// TwinCAT 3 PLC project IDPLC
// ProgramVersion: 3.1.4024.12
// libraries:
//   Recipe Management, * (System)
//   Tc2_Drive, * (Beckhoff Automation GmbH)
//   Tc2_EtherCAT, * (Beckhoff Automation GmbH)
//   Tc2_Math, * (Beckhoff Automation GmbH)
//   Tc2_MC2, * (Beckhoff Automation GmbH)
//   Tc2_ModbusSrv, * (Beckhoff Automation GmbH)
//   Tc2_NC, * (Beckhoff Automation GmbH)
//   Tc2_NcDrive, * (Beckhoff Automation GmbH)
//   Tc2_Standard, * (Beckhoff Automation GmbH)
//   Tc2_System, * (Beckhoff Automation GmbH)
//   Tc2_Utilities, * (Beckhoff Automation GmbH)
//   Tc3_Module, * (Beckhoff Automation GmbH)
//   VisuDialogs, * (System)
// project tree:
//   DUTs/ DUT.TcDUT (not stored), DUT_SENSOR_DATAS_1.TcDUT (not stored), DUT_SENSOR_DATAS_h1.TcDUT, DUT_SENSOR_DATAS_h2.TcDUT, DUT_SENSOR_DATAS_h3.TcDUT, DUT_SENSOR_DATAS_h4.TcDUT, DUT_SENSOR_DATAS_h5.TcDUT, DUT_SENSOR_DATAS_h6.TcDUT, DUT_SENSOR_DATAS_h7.TcDUT, DUT_SENSOR_DATAS_h8.TcDUT, DUT_SENSOR_DATAS_8.TcDUT (not stored), DUT_SENSOR_DATAS_2.TcDUT (not stored), DUT_SENSOR_DATAS_3.TcDUT (not stored), DUT_SENSOR_DATAS_4.TcDUT (not stored), DUT_SENSOR_DATAS_5.TcDUT (not stored), DUT_SENSOR_DATAS_6.TcDUT (not stored), DUT_SENSOR_DATAS_7.TcDUT (not stored), IEEE754_Convert.TcDUT, Struct_M_Compensation.TcDUT (not stored), Struct_M_Gap2Coil.TcDUT, Struct_M_lakeshore.TcDUT (not stored), ST_P180.TcDUT (not stored), ST_P183.TcDUT (not stored), ST_P182.TcDUT (not stored)
//   / GlobalTextList.TcGTLO, PlcTask.TcTTO (not stored), RecipeManager.TcRMO (not stored), Task_Safe.TcTTO, 视图管理器.TcVMO (not stored)
//   GVLs/ Global_Variables.TcGVL, Variable_Configuration.TcGVL (not stored)
//   POUs/0.UserMode/ F_GetSysTime.TcPOU (not stored), UserMode.TcPOU
//   POUs/1.CarrierMode/GapMode/ BCGapMode.TcPOU, GapMode.TcPOU
//   POUs/1.CarrierMode/SingleCarrierMode/ SingleCarrierMode.TcPOU
//   POUs/2.SingleMotorMode/DebugMode/ DebugMode.TcPOU
//   POUs/2.SingleMotorMode/TaperMode/ TaperMode.TcPOU
//   POUs/CoilControl/ PS1.TcPOU, PS3.TcPOU, PS2.TcPOU
//   POUs/CommonFB/ExternFB/ FB_LedShow.TcPOU (not stored), FB_PlcEmergencyStop.TcPOU (not stored)
//   POUs/CommonFB/MainFB/ FB_CoupleAxis.TcPOU, FB_DecoupleAxis.TcPOU, FB_Move.TcPOU, FB_Power.TcPOU, FB_SetAxisPosition.TcPOU, FB_SetMotorAxisPosition.TcPOU, FB_Stop.TcPOU
//   POUs/ MAIN.TcPOU
//   POUs/MainPRG/ FB_CheckCoupleStatus.TcPOU (not stored)
//   POUs/TiltSensor/ FB_Simple_MovingAvg.TcPOU, SAFE.TcPOU
//   VISUs/ Visualization.TcVIS

CONFIGURATION IDPLC
    RESOURCE PLC ON TwinCAT3
        TASK Task_Safe(INTERVAL := T#1ms, PRIORITY := 1);
        PROGRAM SAFE WITH Task_Safe : SAFE;
    END_RESOURCE
END_CONFIGURATION

// ---- DUTs/DUT_SENSOR_DATAS_h1.TcDUT
TYPE DUT_SENSOR_DATAS_h1 :
UNION
	data_lreal:REAL;
	data_byte:ARRAY[0..3] OF BYTE;
END_UNION
END_TYPE

// ---- DUTs/DUT_SENSOR_DATAS_h2.TcDUT
TYPE DUT_SENSOR_DATAS_h2 :
UNION
	data_lreal:REAL;
	data_byte:ARRAY[0..3] OF BYTE;
END_UNION
END_TYPE

// ---- DUTs/DUT_SENSOR_DATAS_h3.TcDUT
TYPE DUT_SENSOR_DATAS_h3 :
UNION
	data_lreal:REAL;
	data_byte:ARRAY[0..3] OF BYTE;
END_UNION
END_TYPE

// ---- DUTs/DUT_SENSOR_DATAS_h4.TcDUT
TYPE DUT_SENSOR_DATAS_h4 :
UNION
	data_lreal:REAL;
	data_byte:ARRAY[0..3] OF BYTE;
END_UNION
END_TYPE

// ---- DUTs/DUT_SENSOR_DATAS_h5.TcDUT
TYPE DUT_SENSOR_DATAS_h5 :
UNION
	data_lreal:REAL;
	data_byte:ARRAY[0..3] OF BYTE;
END_UNION
END_TYPE

// ---- DUTs/DUT_SENSOR_DATAS_h6.TcDUT
TYPE DUT_SENSOR_DATAS_h6 :
UNION
	data_lreal:REAL;
	data_byte:ARRAY[0..3] OF BYTE;
END_UNION
END_TYPE

// ---- DUTs/DUT_SENSOR_DATAS_h7.TcDUT
TYPE DUT_SENSOR_DATAS_h7 :
UNION
	data_lreal:REAL;
	data_byte:ARRAY[0..3] OF BYTE;
END_UNION
END_TYPE

// ---- DUTs/DUT_SENSOR_DATAS_h8.TcDUT
TYPE DUT_SENSOR_DATAS_h8 :
UNION
	data_lreal:REAL;
	data_byte:ARRAY[0..3] OF BYTE;
END_UNION
END_TYPE

// ---- DUTs/IEEE754_Convert.TcDUT
TYPE IEEE754_Convert :
UNION
	data_float:REAL;
	data_word:ARRAY[0..1] OF WORD;
END_UNION
END_TYPE

// ---- DUTs/Struct_M_Gap2Coil.TcDUT
TYPE Struct_M_Gap2Coil :
STRUCT
	Gap:LREAL;
	CoilCurrent:LREAL;
END_STRUCT
END_TYPE

// ---- GVLs/Global_Variables.TcGVL
//{attribute 'Tc2GvlVarNames'}
VAR_GLOBAL
(*IDControl Ready*)
	IDControlReady:BOOL;
(*Maintenance Mode*)
	MaintenanceMode:BOOL;
	MaintenanceModeLed:BOOL;
(*RecipeDescription*)
	RecipeSavedDate:STRING;
	RecipeDescription:STRING;
(*key Command*)
	btn_Power:BOOL;
	btn_PowerOn: BOOL;
	btn_PowerOff: BOOL;
(*Reset*)
	btn_Reset:BOOL;
(*ModeStatus*)
	ModeStatus:INT;
(*Error Massage*)
	Error:BOOL;
	ErrorID:DINT;
	ErrorDescription:STRING;
(*加载配方参数*)
	LoadRecipeParameters:BOOL;
	loadParametersDone:BOOL;
(*Max Velocity Global*)
	MaxVelocityGlobalVelocity : LREAL;
(*设置光栅bias done *)	
	PositionBiasDone:BOOL;
(*回程差*)
	HysteresisError:LREAL;
(*Drive Status*)
	DriveStatus:DINT;//1:Drive Ready;2:Axis is in operation;0:Others
(*光栅漂移误差阈值*)
	LEDriftErrorThreshold:LREAL:=0.001;
(*Lag Distance threshold*)
	PosDiff_LeftTopLin: LREAL:=0.5;
	PosDiff_RightTopLin:LREAL:=0.5;
	PosDiff_LeftBottomLin:LREAL:=0.5;
	PosDiff_RightBottomLin:LREAL:=0.5;
(*UserMode Threshold*)
	Threshold_UserTopPos: LREAL:=0.5;
	Threshold_UserBottomPos: LREAL:=0.5;
	Threshold_UserLeftPos: LREAL:=0.5;
	Threshold_UserRightPos: LREAL:=0.5;
	Threshold_UserTopVelo: LREAL:=0.5;
	Threshold_UserBottomVelo: LREAL:=0.5;
	Threshold_UserLeftVelo: LREAL:=0.5;
	Threshold_UserRightVelo: LREAL:=0.5;
	//
	Range_UserTaperPos:LREAL:=4.01;
	Range_UserTaperVelo:LREAL:=1.01;
	//Diff_TaperLeftPos:LREAL:=0.01;
	//Diff_TaperLeftVelo:LREAL:=0.2;
	//Diff_TaperRightPos:LREAL:=0.05;
	//Diff_TaperRightVelo:LREAL:=0.5;
	//Taper_BeyondRangePositive:BOOL;
	//Diff_TaperTopPos:LREAL:=0.05;
	//Diff_TaperBottomPos:LREAL:=0.05;
	//Taper_BeyondRangeNegtive:BOOL;
(*BCGap Threshold*)
	Threshold_BCTopPos: LREAL:=0.5;
	Threshold_BCBottomPos: LREAL:=0.5;
	Threshold_BCLeftPos: LREAL:=0.5;
	Threshold_BCRightPos: LREAL:=0.5;
	Threshold_BCTopVelo: LREAL:=0.5;
	Threshold_BCBottomVelo: LREAL:=0.5;
	Threshold_BCLeftVelo: LREAL:=0.5;
	Threshold_BCRightVelo: LREAL:=0.5;
(*DebugMode Threshold*)
	Threshold_TopPos_Debug: LREAL:=4;
	Threshold_BottomPos_Debug: LREAL:=4;
	Threshold_LeftPos_Debug: LREAL:=4;
	Threshold_RightPos_Debug: LREAL:=4;
	//单轴目标位置和当前位置之差，阈值
	Threshold_LeftTopPos_Debug: LREAL:=0.4;	
	Threshold_RightTopPos_Debug: LREAL:=0.4;
	Threshold_LeftBottomPos_Debug: LREAL:=0.4;
	Threshold_RightBottomPos_Debug: LREAL:=0.4;
(*Taper Mode Threshold*)
	Range_TaperPos:LREAL:=5.01;
	Range_TaperVelo:LREAL:=1.01;
	Threshold_TaperLeftPos:LREAL:=0.01;
	Threshold_TaperLeftVelo:LREAL:=0.2;
	Threshold_TaperRightPos:LREAL:=0.05;
	Threshold_TaperRightVelo:LREAL:=0.5;
	Taper_BeyondRangePositive:BOOL;
	Threshold_TaperTopPos:LREAL:=0.05;
	Threshold_TaperBottomPos:LREAL:=0.05;
	Taper_BeyondRangeNegtive:BOOL;
(*SingleCarrierMode threshold*)
	Threshold_TopPos_SingleCarrier: LREAL:=2;
	Threshold_BottomPos_SingleCarrier: LREAL:=2;
	Threshold_LeftPos_SingleCarrier: LREAL:=2;
	Threshold_RightPos_SingleCarrier: LREAL:=2;
	Threshold_TopVelo_SingleCarrier: LREAL:=2;
	Threshold_BottomVelo_SingleCarrier: LREAL:=2;
	Threshold_LeftVelo_SingleCarrier: LREAL:=2;
	Threshold_RightVelo_SingleCarrier: LREAL:=2;
(*Compensation Value*)
	(*Moving or notmoving*)
	moveStatusLeftTop: BOOL;
	moveStatusRightTop: BOOL;
	moveStatusLeftBottom: BOOL;
	moveStatusRightBottom: BOOL;
	moveStatusAllAxis: BOOL;
	moveStatusAnyAxis: BOOL;
	moveStatusGap:BOOL;
	moveStatusTaper:BOOL;
(*Moving or notmoving-Motor*)
	moveStatusLeftTopMotor: BOOL;
	moveStatusRightTopMotor: BOOL;
	moveStatusLeftBottomMotor: BOOL;
	moveStatusRightBottomMotor: BOOL;
	moveStatusAllAxisMotor: BOOL;
	moveStatusAnyAxisMotor: BOOL;
	(*input protection*)
	//
	min_UserGapPositionNew:LREAL:=10;
	max_UserGapPositionNew:LREAL:=200;
	inRange_UserGapPositionNew:BOOL;
	//LE protection position
	min_UserLEProtectionGapPosition:LREAL;
	min_ThresholdGapSoft2LEProtection:LREAL;
	max_UserLEProtectionGapPosition:LREAL;
	max_ThresholdGapSoft2LEProtection:LREAL;
	//
	min_UserGapVelocityNew:LREAL:=0;
	max_UserGapVelocityNew:LREAL:=2;
	inRange_UserGapVelocityNew:BOOL;
	//
	min_UserTaperPositionNew: LREAL:=0;;
	max_UserTaperPositionNew: LREAL:=1;
	inRange_UserTaperPositionNew: BOOL;
	//
	min_UserTaperVelocityNew: LREAL:=0;
	max_UserTaperVelocityNew: LREAL:=1;
	inRange_UserTaperVelocityNew: BOOL;

	M_Compensation:ARRAY[1..18] OF Struct_M_Compensation
:=[
(Encoder:=0,	LeftTop:=0,	RightTop:=0,		LeftBottom:=0,	RightBottom:=0,	InRange:=FALSE),
(Encoder:=5.5,	LeftTop:=5.5,	RightTop:=5.5,	LeftBottom:=5.5,	RightBottom:=5.5,	InRange:=FALSE),
(Encoder:=6.0,	LeftTop:=6.0,	RightTop:=6.0,	LeftBottom:=6.0,	RightBottom:=6.0,	InRange:=FALSE),
(Encoder:=6.5,	LeftTop:=6.5,	RightTop:=6.5,	LeftBottom:=6.5,	RightBottom:=6.5,	InRange:=FALSE),
(Encoder:=7.5,	LeftTop:=7.5,	RightTop:=7.5,	LeftBottom:=7.5,	RightBottom:=7.5,	InRange:=FALSE),
(Encoder:=8.5,	LeftTop:=8.5,	RightTop:=8.5,	LeftBottom:=8.5,	RightBottom:=8.5,	InRange:=FALSE),
(Encoder:=9.5,	LeftTop:=9.5,	RightTop:=9.5,	LeftBottom:=9.5,	RightBottom:=9.5,	InRange:=FALSE),
(Encoder:=10.5,	LeftTop:=10.5,	RightTop:=10.5,	LeftBottom:=10.5,	RightBottom:=10.5,		InRange:=FALSE),
(Encoder:=11.5,	LeftTop:=11.5,	RightTop:=11.5,	LeftBottom:=11.5,	RightBottom:=11.5,		InRange:=FALSE),
(Encoder:=30.0,	LeftTop:=30.0,	RightTop:=30.0,	LeftBottom:=30.0,	RightBottom:=30.0,		InRange:=FALSE),
(Encoder:=100.0,	LeftTop:=100.0,	RightTop:=100.0,	LeftBottom:=100.0,	RightBottom:=100.0,		InRange:=FALSE),
(Encoder:=110.0,	LeftTop:=110.0,	RightTop:=110.0,	LeftBottom:=110.0,	RightBottom:=110.0,		InRange:=FALSE),
(Encoder:=120.0,	LeftTop:=120.0,	RightTop:=120.0,	LeftBottom:=120.0,	RightBottom:=120.0,		InRange:=FALSE),
(Encoder:=130.0,	LeftTop:=130.0,	RightTop:=130.0,	LeftBottom:=130.0,	RightBottom:=130.0,		InRange:=FALSE),
(Encoder:=140.0,	LeftTop:=140.0,	RightTop:=140.0,	LeftBottom:=140.0,	RightBottom:=140.0,		InRange:=FALSE),
(Encoder:=150.0,	LeftTop:=150.0,	RightTop:=150.0,	LeftBottom:=150.0,	RightBottom:=150.0,		InRange:=FALSE),
(Encoder:=160.0,	LeftTop:=160.0,	RightTop:=160.0,	LeftBottom:=160.0,	RightBottom:=160.0,		InRange:=FALSE),
(Encoder:=3000.001,	LeftTop:=3000.001,	RightTop:=3000.001,		LeftBottom:=3000.001,	RightBottom:=3000.001,	InRange:=FALSE)];

(*simulation OR NOT*)
	simulation:BOOL;
(*USELinearEncoeder*)
	USELinearEncoder:BOOL:=TRUE;
(*restartTwinCAT*)
	m_restartTC:BOOL;
	m_simpleRestartTC:BOOL;
(*Plc_EmergencyStop *)
	Plc_EmergencyStop  AT %Q*:BOOL:=TRUE;
(*硬急停*)
	Hardware_EmergencyStop :BOOL:=TRUE;
(*LED*)
	Led_Run  AT %Q*:BOOL;
	Led_Error  AT %Q*:BOOL;
(*LimitSwitch*)
	LS_LeftTop_Far  :BOOL;
	LS_LeftTop_Near  :BOOL;
	LS_RightTop_Far  :BOOL;
	LS_RightTop_Near  :BOOL;
	LS_LeftBottom_Far  :BOOL;
	LS_LeftBottom_Near  :BOOL;
	LS_RightBottom_Far :BOOL;
	LS_RightBottom_Near  :BOOL;
	Unreach_LS_Far:BOOL;
	Unreach_LS_Near:BOOL;
(*kill switch*)
	KS_LeftTop_Far_Contact1:BOOL;
	KS_LeftTop_Far_Contact2:BOOL;
	KS_RightTop_Far_Contact1:BOOL;
	KS_RightTop_Far_Contact2:BOOL;
	KS_LeftBottom_Far_Contact1:BOOL;
	KS_LeftBottom_Far_Contact2:BOOL;
	KS_RightBottom_Far_Contact1:BOOL;
	KS_RightBottom_Far_Contact2:BOOL;
	
	KS_LeftTop_Near_Contact1:BOOL;
	KS_LeftTop_Near_Contact2:BOOL;
	KS_RightTop_Near_Contact1:BOOL;
	KS_RightTop_Near_Contact2:BOOL;
	KS_LeftBottom_Near_Contact1:BOOL;
	KS_LeftBottom_Near_Contact2:BOOL;
	KS_RightBottom_Near_Contact1:BOOL;
	KS_RightBottom_Near_Contact2:BOOL;
(*E-STOP*)
	KS_CabinetEmergency_contact1:BOOL;
	KS_CabinetEmergency_contact2:BOOL;
	KS_handEmergency1_Contact1:BOOL;
	KS_handEmergency1_Contact2:BOOL;
	KS_handEmergency2_Contact1:BOOL;
	KS_handEmergency2_Contact2:BOOL;
	KS_softEmergency2_Contact:BOOL;
(*aixs_ref*)
	LeftTopLin: axis_ref;
	RightTopLin:axis_ref;
	LeftBottomLin:axis_ref;
	RightBottomLin:axis_ref;
(*aixs_ref-motor*)
	LeftTopMotor: axis_ref;
	RightTopMotor:axis_ref;
	LeftBottomMotor:axis_ref;
	RightBottomMotor:axis_ref;
(*axis Position*)
	{attribute:'TcAnalytics'}
	Pos_LeftTopLin: LREAL;
	{attribute:'TcAnalytics'}
	Pos_RightTopLin:LREAL;
	{attribute:'TcAnalytics'}
	Pos_LeftBottomLin:LREAL;
	{attribute:'TcAnalytics'}
	Pos_RightBottomLin:LREAL;
(*axis Position-motor*)
	Pos_LeftTopMotor: LREAL;
	Pos_RightTopMotor:LREAL;
	Pos_LeftBottomMotor:LREAL;
	Pos_RightBottomMotor:LREAL;
(*axis Position-Delta*)
	DeltaPos_LeftTop: LREAL;
	DeltaPos_RightTop:LREAL;
	DeltaPos_LeftBottom:LREAL;
	DeltaPos_RightBottom:LREAL;
(*axis Position-Threshold*)
	ThresholdDeltaPos_LeftTop: LREAL:=0.2;
	ThresholdDeltaPos_RightTop:LREAL:=0.2;
	ThresholdDeltaPos_LeftBottom:LREAL:=0.2;
	ThresholdDeltaPos_RightBottom:LREAL:=0.2;
(*axis Velocity*)
	Velo_LeftTopLin: LREAL;
	Velo_RightTopLin:LREAL;
	Velo_LeftBottomLin:LREAL;
	Velo_RightBottomLin:LREAL;
(*axis Velocity-motor*)
	Velo_LeftTopMotor: LREAL;
	Velo_RightTopMotor:LREAL;
	Velo_LeftBottomMotor:LREAL;
	Velo_RightBottomMotor:LREAL;
(*axis Velocity-Delta*)
	DeltaVelo_LeftTop: LREAL;
	DeltaVelo_RightTop:LREAL;
	DeltaVelo_LeftBottom:LREAL;
	DeltaVelo_RightBottom:LREAL;
(*axis Velocity-ThresholdDelta*)
	ThresholdDeltaVelo_LeftTop: LREAL:=0.1;
	ThresholdDeltaVelo_RightTop:LREAL:=0.1;
	ThresholdDeltaVelo_LeftBottom:LREAL:=0.1;
	ThresholdDeltaVelo_RightBottom:LREAL:=0.1;
(*axis Torque-motor*)
	Torque_LeftTopLin: LREAL;
	Torque_RightTopLin:LREAL;
	Torque_LeftBottomLin:LREAL;
	Torque_RightBottomLin:LREAL;
(*axis Torque-motor*)
	Torque_LeftTopMotor: LREAL;
	Torque_RightTopMotor:LREAL;
	Torque_LeftBottomMotor:LREAL;
	Torque_RightBottomMotor:LREAL;
(*axis Torque-Delta*)
	DeltaTorque_LeftTop: LREAL;
	DeltaTorque_RightTop:LREAL;
	DeltaTorque_LeftBottom:LREAL;
	DeltaTorque_RightBottom:LREAL;
(*Lag Distance*)
	PosDiff_LeftTopLin_actual: LREAL;
	PosDiff_RightTopLin_actual:LREAL;
	PosDiff_LeftBottomLin_actual:LREAL;
	PosDiff_RightBottomLin_actual:LREAL;
(*Lag Distance-Motor*)
	PosDiff_LeftTopMotor_actual: LREAL;
	PosDiff_RightTopMotor_actual:LREAL;
	PosDiff_LeftBottomMotor_actual:LREAL;
	PosDiff_RightBottomMotor_actual:LREAL;
(*Delta LagDistance*)
	DeltaPosDiff_LeftTop_actual: LREAL;
	DeltaPosDiff_RightTop_actual:LREAL;
	DeltaPosDiff_LeftBottom_actual:LREAL;
	DeltaPosDiff_RightBottom_actual:LREAL;
(********************Gap Mode*************************)
(**)
	GapPositionActual:LREAL;
	GapVelocityActual:LREAL;
	GapMoveIndicator:DINT:=0;
	(*1=OPEN;0=NOTMOVE;-1=CLOSE*)
(******************Taper Mode**************************)
(*Taper*)
	TaperPositionActual:LREAL;
	TaperVelocityActual:LREAL;
	TaperMoveIndicator:DINT:=0;
	(*1=OPEN;0=NOTMOVE;-1=CLOSE*)
(*****************singleCarrier Mode*******************************)
(**)
	TopPositionActual:LREAL;
	TopVelocityActual:LREAL;
	BottomPositionActual:LREAL;
	BottomVelocityActual:LREAL;
	TopMoveIndicator:DINT:=0;
	(*1=OPEN;0=NOTMOVE;-1=CLOSE*)
	BottomMoveIndicator:DINT:=0;
	(*1=OPEN;0=NOTMOVE;-1=CLOSE*)
(******************DebugMode & BCGapMode*****************************)
	LeftTopLinMoveIndicator:DINT:=0;
	(*1=OPEN;0=NOTMOVE;-1=CLOSE*)
	LeftBottomLinMoveIndicator:DINT:=0;
	(*1=OPEN;0=NOTMOVE;-1=CLOSE*)
	RightTopLinMoveIndicator:DINT:=0;
	(*1=OPEN;0=NOTMOVE;-1=CLOSE*)
	RightBottomLinMoveIndicator:DINT:=0;
	(*1=OPEN;0=NOTMOVE;-1=CLOSE*)
(******************Gap&SingleCarrier***********************************)
	Diff_TopPos_actual: LREAL;
	Diff_BottomPos_actual: LREAL;
	Diff_LeftPos_actual: LREAL;
	Diff_RightPos_actual: LREAL;
	Diff_TopVelo_actual:  LREAL;
	Diff_BottomVelo_actual: LREAL;
	Diff_LeftVelo_actual: LREAL;
	Diff_RightVelo_actual:  LREAL;

(******************BCGap Mode***********************************)
	Diff_BCTopPos_actual: LREAL;
	Diff_BCBottomPos_actual: LREAL;
	Diff_BCLeftPos_actual: LREAL;
	Diff_BCRightPos_actual: LREAL;
	Diff_BCTopVelo_actual:  LREAL;
	Diff_BCBottomVelo_actual: LREAL;
	Diff_BCLeftVelo_actual: LREAL;
	Diff_BCRightVelo_actual:  LREAL;
(******************UserMode*********************)
	Diff_UserTopPos_actual: LREAL;
	Diff_UserBottomPos_actual: LREAL;
	Diff_UserLeftPos_actual: LREAL;
	Diff_UserRightPos_actual: LREAL;
	Diff_UserTopVelo_actual:  LREAL;
	Diff_UserBottomVelo_actual: LREAL;
	Diff_UserLeftVelo_actual: LREAL;
	Diff_UserRightVelo_actual:  LREAL;
	//ID taper Mode
	TaperFunctionSolidOn:BOOL;//该ID是否有taper需求，taper总开关，只在参数表生效
	TaperOrNot:BOOL;//ID taper功能开关，入口电机不动，出口电机动
	UserTaperPositionActual:LREAL;
	UserTaperVelocityActual:LREAL;
(***********************Power status and couple statatus***********************)
	st_Power:BOOL;
	st_Couple:DINT;
(************************FB***********************)
	FB_Power:FB_Power;
	FB_PlcEmergencyStop: FB_PlcEmergencyStop;
	FB_CheckCoupleStatus:FB_CheckCoupleStatus;
	FB_Move:FB_Move;
	FB_Stop:FB_Stop;
	FB_DecoupleAxis:FB_DecoupleAxis;
	FB_CoupleAxis: FB_CoupleAxis;
(********************²¹³¥GapÄ£Ê½£¬µ¥Öá²¹³¥Êý¾Ý************************)
	(*ÊÇ·ñ²¹³¥*)
	USE_SingleAxis_Compensation:BOOL:=TRUE;
	Mdut:ARRAY[1..2] OF DUT:=
	[(Encoder:=2.0,	LeftTop:=2.3000),
	(Encoder:=2.0,	LeftTop:=2.3000)];


	M_CompensationNumber:INT;
	M_DisplayNumber:INT;
	(*Conpensation Position Target*)
	LeftTopLinPositionNew:LREAL;
	LeftBottomLinPositionNew:LREAL;
	RightTopLinPositionNew:LREAL;
	RightBottomLinPositionNew:LREAL;
	(*考虑到回程差后，运动到临时位置*)
	LeftTopLinPositionNew_temporary :LREAL;
	LeftBottomLinPositionNew_temporary:LREAL;
	RightTopLinPositionNew_temporary:LREAL;
	RightBottomLinPositionNew_temporary:LREAL;
	(*Display Position*)
	LeftTopLinPositionDisplay:LREAL;
	LeftBottomLinPositionDisplay:LREAL;
	RightTopLinPositionDisplay:LREAL;
	RightBottomLinPositionDisplay:LREAL;
	(*Display Velocity*)
	LeftTopLinVelocityDisplay:LREAL;
	LeftBottomLinVelocityDisplay:LREAL;
	RightTopLinVelocityDisplay:LREAL;
	RightBottomLinVelocityDisplay:LREAL;
	(*temperature sensors*)
	thermocouple AT %I*:ARRAY[1..12]OF  DINT;
	shieldPt100  AT %I*:ARRAY[1..12]OF INT;
	thermocouple_Celsius:ARRAY[1..12]OF  LREAL;
	shieldPt100_Celsius  :ARRAY[1..12]OF LREAL;
	huoer_Celsius AT %I* :ARRAY[1..3]OF INT;
	(**)
	lakeshorePt100  AT %I*:ARRAY[1..12]OF INT;(*16*×èÖµ*)
	lakeshorePt100_Resistance :ARRAY[1..12]OF LREAL;(*ÉãÊÏÎÂ¶È*)
	lakeshorePt100_Celsius  :ARRAY[1..12]OF LREAL;(*ÉãÊÏÎÂ¶È*)
	temperatureCompensationValue:LREAL:=6;
	testSensors  AT %I*:ARRAY[1..4]OF INT;

(*Test No.184*)
	Struct_M_lakeshore_168:ARRAY[1..52] OF Struct_M_lakeshore:=[(Temperature:=-255.02072961,	Resistance:=19394.22709513),
														       (Temperature:=-254.05045152,	Resistance:=17654.92429047),
														       (Temperature:=-253.07744087,	Resistance:=16151.62683151),
														       (Temperature:=-252.00959324,	Resistance:=14730.57326945),
														       (Temperature:=-250.42495220,	Resistance:=12968.55015283),
														       (Temperature:=-248.82081761,	Resistance:=11509.89960915),
														       (Temperature:=-247.21174565,	Resistance:=10296.55197911),
														       (Temperature:=-245.58891366,	Resistance:=9270.75571767),
														       (Temperature:=-243.96558907,	Resistance:=8400.62569432),
														       (Temperature:=-242.14354329,	Resistance:=7573.26483503),
														       (Temperature:=-240.02689351,	Resistance:=6767.17126789),
														       (Temperature:=-237.01618411,	Resistance:=5838.58514549),
														       (Temperature:=-234.00593745,	Resistance:=5101.58555065),
														       (Temperature:=-230.99752410,	Resistance:=4505.18214539),
														       (Temperature:=-228.00173193,	Resistance:=4017.09732257),
														       (Temperature:=-224.99947745,	Resistance:=3609.02040601),
														       (Temperature:=-223.00692641,	Resistance:=3374.28026471),
														       (Temperature:=-218.01660226,	Resistance:=2884.61719537),
														       (Temperature:=-213.02574325,	Resistance:=2501.58514940),
														       (Temperature:=-208.03560884,	Resistance:=2195.64012040),
														       (Temperature:=-203.04420176,	Resistance:=1946.81103230),
														       (Temperature:=-198.05275449,	Resistance:=1741.06206884),
														       (Temperature:=-193.06103279,	Resistance:=1568.92560629),
														       (Temperature:=-188.06248282,	Resistance:=1422.92395120),
														       (Temperature:=-183.06714354,	Resistance:=1298.17958491),
														       (Temperature:=-178.06870827,	Resistance:=1190.47468069),
														       (Temperature:=-173.07068956,	Resistance:=1096.60468916),
														       (Temperature:=-163.08053594,	Resistance:=942.07281950),
														       (Temperature:=-153.08718985,	Resistance:=820.42837839),
														       (Temperature:=-143.08487641,	Resistance:=722.56760466),
														       (Temperature:=-133.08398781,	Resistance:=642.67848926),
														       (Temperature:=-123.08745222,	Resistance:=576.45895597),
														       (Temperature:=-113.09120089,	Resistance:=520.90762376),
														       (Temperature:=-103.09942915,	Resistance:=473.74837218),
														       (Temperature:=-93.10598968,		Resistance:=433.38294834),
														       (Temperature:=-83.10392915,		Resistance:=398.41968464),
														       (Temperature:=-73.10228709,		Resistance:=368.09301028),
														       (Temperature:=-63.10299621,		Resistance:=341.43424414),
														       (Temperature:=-53.11519681,		Resistance:=318.02847824),
														       (Temperature:=-43.10742807	,	Resistance:=297.22485607),
														       (Temperature:=-33.10726812,		Resistance:=278.69871028),
														       (Temperature:=-23.11858134,		Resistance:=262.15834948),
														       (Temperature:=-13.10195090,		Resistance:=247.23616978),
														       (Temperature:=-3.11184252,		Resistance:=233.79708047),
														       (Temperature:=6.89903472,		Resistance:=221.61300733),
														       (Temperature:=16.89346621,		Resistance:=210.54967929),
														       (Temperature:=26.90358952,		Resistance:=200.45587628),
														       (Temperature:=36.88287604,		Resistance:=191.25204791),
														       (Temperature:=41.88872196,		Resistance:=186.92616816),
														       (Temperature:=46.88480694,		Resistance:=182.78432099),
														       (Temperature:=52.87776550,		Resistance:=178.06184409),
														       (Temperature:=56.87370113,		Resistance:=175.01081354)];

(*
Struct_M_lakeshore_168:ARRAY[1..52] OF Struct_M_lakeshore:=(Temperature:=-255.02148584,	Resistance:=17467.51361429),
														       (Temperature:=-254.05229765,	Resistance:=15920.82205731),
														       (Temperature:=-253.07582822,	Resistance:=14578.50586503),
														       (Temperature:=-252.01029408,	Resistance:=13314.83293750),
														       (Temperature:=-250.42593953,	Resistance:=11741.46150061),
														       (Temperature:=-248.82114671,	Resistance:=10435.92048251),
														       (Temperature:=-247.21093179,	Resistance:=9348.73725539),
														       (Temperature:=-245.58869114,	Resistance:=8428.36508630),
														       (Temperature:=-243.96317077,	Resistance:=7645.95382882),
														       (Temperature:=-242.14282659,	Resistance:=6901.52980185),
														       (Temperature:=-240.02565306,	Resistance:=6174.70288700),
														       (Temperature:=-237.01772619,	Resistance:=5337.15935418),
														       (Temperature:=-234.00641032,	Resistance:=4669.94432605),
														       (Temperature:=-230.99638631,	Resistance:=4129.44762482),
														       (Temperature:=-228.00091359,	Resistance:=3686.25091590),
														       (Temperature:=-225.00020456,	Resistance:=3315.69773718),
														       (Temperature:=-223.00791577,	Resistance:=3102.03825436),
														       (Temperature:=-218.01784455,	Resistance:=2655.95765650),
														       (Temperature:=-213.02820409,	Resistance:=2306.30469335),
														       (Temperature:=-208.03707086,	Resistance:=2026.68631979),
														       (Temperature:=-203.04413996,	Resistance:=1798.75031171),
														       (Temperature:=-198.05551086,	Resistance:=1610.35975891),
														       (Temperature:=-193.06273927,	Resistance:=1452.39526661),
														       (Temperature:=-188.05883288,	Resistance:=1318.25592597),
														       (Temperature:=-183.06258538,	Resistance:=1203.56234118),
														       (Temperature:=-178.06718279,	Resistance:=1104.51148216),
														       (Temperature:=-173.07249199,	Resistance:=1018.20332165),
														       (Temperature:=-163.08375191,	Resistance:=875.68114167),
														       (Temperature:=-153.08708895,	Resistance:=763.40014611),
														       (Temperature:=-143.08456026,	Resistance:=673.01413079),
														       (Temperature:=-133.08511977,	Resistance:=599.14558137),
														       (Temperature:=-123.08749266,	Resistance:=537.87435730),
														       (Temperature:=-113.09351200,	Resistance:=486.39730699),
														       (Temperature:=-103.10083499,	Resistance:=442.70701049),
														       (Temperature:=-93.10681179,		Resistance:=405.24490154),
														       (Temperature:=-83.10668364,		Resistance:=372.85251196),
														       (Temperature:=-73.10424427,		Resistance:=344.62377216),
														       (Temperature:=-63.10525050,		Resistance:=319.91272482),
														       (Temperature:=-53.11631884,		Resistance:=298.14326645),
														       (Temperature:=-43.10919062	,	Resistance:=278.79776489),
														       (Temperature:=-33.10718139,		Resistance:=261.57224548),
														       (Temperature:=-23.12143823,		Resistance:=246.17864217),
														       (Temperature:=-13.10564070,		Resistance:=232.27707124),
														       (Temperature:=-3.11271856,		Resistance:=219.77787693),
														       (Temperature:=6.89876028,		Resistance:=208.41568062),
														       (Temperature:=16.88935188,		Resistance:=198.10158580),
														       (Temperature:=26.89992337,		Resistance:=188.70405160),
														       (Temperature:=36.88110394,		Resistance:=180.10572832),
														       (Temperature:=41.88616228,		Resistance:=176.08361784),
														       (Temperature:=46.88372409,		Resistance:=172.21346348),
														       (Temperature:=52.87452959,		Resistance:=167.80352164),
														       (Temperature:=56.87233822,		Resistance:=164.96790544);
*)

(******RS232************)
	//			: ComBuffer;	(* Receive data buffer; used with all receive function blocks *)
	//TxBufferEL			: ComBuffer;	(* Transmit data buffer; used with all receive function blocks *)

	(*ColiControl Function*)
	(*Use in HALF *)
	CoilControlFunction:BOOL:=FALSE;
	(*add Beamline taper 模式，入口和出口电机都运动，保持中心gap不变*)
	//3种模式划分：
	NormalGapMode:BOOL;
	IDTaperMode:BOOL;
	BLTaperMode:BOOL;
	//BLtaper相关参数
	BLTaperOrNot:BOOL;//ID taper功能开关，入口电机不动，出口电机动
	BLUserTaperPositionActual:LREAL;
	BLUserTaperVelocityActual:LREAL;
		//
	min_BLUserTaperPositionNew: LREAL:=0;;
	max_BLUserTaperPositionNew: LREAL:=1;
	inRange_BLUserTaperPositionNew: BOOL;
	//
	min_BLUserTaperVelocityNew: LREAL:=0;
	max_BLUserTaperVelocityNew: LREAL:=1;
	inRange_BLUserTaperVelocityNew: BOOL;
END_VAR

// ---- POUs/TiltSensor/SAFE.TcPOU
PROGRAM SAFE
VAR
	TiltSensorFunctionOn:BOOL;
	//
	//Top TiltSensor
	//
	TiltSensorTopAngle_INT AT%I*: INT;
	TiltSensorTopAngle_mA: LREAL;
	TileSensorTop_SN:STRING:='TT1026';
	TiltSensorTop_ScaleFactor: LREAL:=0.0596;
	fbMovingAvg_TiltSensorTop : FB_Simple_MovingAvg;
	TiltSensorTop_FilterWindow : INT := 1000;  // 100个周期平均 = 1000ms
	TiltSensorTop_mA_Filter:LREAL;
	TiltSensorTop_mA:LREAL;
	//角度，单位：°
	TiltSensorTopAngle: LREAL;	
	//滤波后角度，单位：°
	TiltSensorTopAngle_Filter: LREAL;
	TileSensorTop_Underrange AT%I*:BOOL;
	TileSensorTop_Overrange AT%I*:BOOL;
	TileSensorTop_Error AT%I*:BOOL;
	TiltSensorTopAngle_mA_Filter: LREAL;
	//TileMotorOffset: REAL;
	//L_Center2Motor: INT:=1375;
	//初始准直零位角度
	TiltSensorTop_InitAngle:LREAL;
	//角度阈值
	TiltSensorTop_GapThreshold:LREAL;
	TiltSensorTop_IDTaperThreshold:LREAL;
	TiltSensorTop_BLTaperThreshold:LREAL;
	//角度与taper的比例
	TaperAndTileTopAngleScale:LREAL;
		//
	//Bottom TiltSensor
	//
	TiltSensorBottomAngle_INT AT%I*: INT;
	TiltSensorBottomAngle_mA: LREAL;
	TileSensorBottom_SN:STRING:='TT1026';
	TiltSensorBottom_ScaleFactor: LREAL:=0.0596;
	fbMovingAvg_TiltSensorBottom : FB_Simple_MovingAvg;
	TiltSensorBottom_FilterWindow : INT := 1000;  // 100个周期平均 = 1000ms
	TiltSensorBottom_mA_Filter:LREAL;
	TiltSensorBottom_mA:LREAL;
	//角度，单位：°
	TiltSensorBottomAngle: LREAL;	
	//滤波后角度，单位：°
	TiltSensorBottomAngle_Filter: LREAL;
	TileSensorBottom_Underrange AT%I*:BOOL;
	TileSensorBottom_Overrange AT%I*:BOOL;
	TileSensorBottom_Error AT%I*:BOOL;
	TiltSensorBottomAngle_mA_Filter: LREAL;
	//TileMotorOffset: REAL;
	//L_Center2Motor: INT:=1375;
	//初始准直零位角度
	TiltSensorBottom_InitAngle:LREAL;
	//角度阈值
	TiltSensorBottom_GapThreshold:LREAL;
	TiltSensorBottom_IDTaperThreshold:LREAL;
	TiltSensorBottom_BLTaperThreshold:LREAL;
	//角度与taper的比例
	TaperAndTileBottomAngleScale:LREAL;
	
	a: LREAL;
END_VAR

//
//Function On/OFF
//
IF NOT TiltSensorFunctionOn THEN
	RETURN;
END_IF
//
//Top TiltSensor
//
TiltSensorTopAngle_mA:=(INT_TO_LREAL(TiltSensorTopAngle_INT)/32767)*16+4;
// 每个PLC周期（10ms）调用一次,移动平均
fbMovingAvg_TiltSensorTop(x := TiltSensorTopAngle_mA,    // 输入原始值
            N := TiltSensorTop_FilterWindow,  // 窗口大小
            rst := FALSE,       // 不复位
            y => TiltSensorTopAngle_mA_Filter);     // 输出平均值
//计算角度
TiltSensorTopAngle_Filter:=DINT_TO_LREAL(LREAL_TO_DINT(((TiltSensorTopAngle_mA_Filter-12)*TiltSensorTop_ScaleFactor+TiltSensorTop_InitAngle)*100000))/100000;//滤波后
TiltSensorTopAngle:=DINT_TO_LREAL(LREAL_TO_DINT(((TiltSensorTopAngle_mA-12)*TiltSensorTop_ScaleFactor+TiltSensorTop_InitAngle)*100000))/100000;//未滤波，原始数据
//计算电机处由于倾斜导致的偏移量，单位毫米
//TileMotorOffset:=L_Center2Motor*2*TAN(TiltSensorAngle_degree*PI / 180);
//阈值触发
IF NormalGapMode THEN
	IF TiltSensorTopAngle>TiltSensorTop_GapThreshold THEN
		ErrorID:=1601;
		Error:=TRUE;
		ErrorDescription:='TiltSensorTopAngle>TiltSensorTop_Threshold';
		FB_PlcEmergencyStop();
		LED_Error:=TRUE;
	END_IF
END_IF
IF IDTaperMode THEN
	IF TiltSensorTopAngle>TiltSensorTop_IDTaperThreshold THEN
		ErrorID:=1602;
		Error:=TRUE;
		ErrorDescription:='TiltSensorTopAngle>TiltSensorTop_IDTaperThreshold';
		FB_PlcEmergencyStop();
		LED_Error:=TRUE;
	END_IF
END_IF
IF BLTaperMode THEN
	IF TiltSensorTopAngle>TiltSensorTop_BLTaperThreshold THEN
		ErrorID:=1603;
		Error:=TRUE;
		ErrorDescription:='TiltSensorTopAngle>TiltSensorTop_BLTaperThreshold';
		FB_PlcEmergencyStop();
		LED_Error:=TRUE;
	END_IF
END_IF
//角度与taper的比例
IF NormalGapMode THEN
	TaperAndTileTopAngleScale:=0;
ELSIF IDTaperMode THEN
	TaperAndTileTopAngleScale:=DINT_TO_LREAL(LREAL_TO_DINT((ATAN((UserMode.UserTaperPositionNew/2)/(2*UserMode.L_Center2Motor))*180/PI)*100000))/100000;
ELSIF BLTaperMode THEN
	TaperAndTileTopAngleScale:=DINT_TO_LREAL(LREAL_TO_DINT((ATAN((UserMode.BLUserTaperPositionNew/4)/(UserMode.L_HalfGirder))*180/PI)*100000))/100000;
END_IF
//超出检测范围处理
IF TileSensorTop_Underrange THEN
	ErrorID:=1604;
	Error:=TRUE;
	ErrorDescription:='TileSensorTop_Underrange';
	//FB_PlcEmergencyStop();
	LED_Error:=TRUE;
ELSE
	ErrorID:=0;
	Error:=FALSE;
	ErrorDescription:='';
	LED_Error:=FALSE;
END_IF
IF TileSensorTop_Overrange THEN
	ErrorID:=1605;
	Error:=TRUE;
	ErrorDescription:='TileSensorTop_Overrange';
	//FB_PlcEmergencyStop();
	LED_Error:=TRUE;
ELSE
	ErrorID:=0;
	Error:=FALSE;
	ErrorDescription:='';
	LED_Error:=FALSE;
END_IF
IF TileSensorTop_Error THEN
	ErrorID:=1606;
	Error:=TRUE;
	ErrorDescription:='TileSensorTop_Error';
	//FB_PlcEmergencyStop();
	LED_Error:=TRUE;
ELSE
	ErrorID:=0;
	Error:=FALSE;
	ErrorDescription:='';
	LED_Error:=FALSE;
END_IF
//
//Bottom TiltSensor
//
TiltSensorBottomAngle_mA:=(INT_TO_LREAL(TiltSensorBottomAngle_INT)/32767)*16+4;
// 每个PLC周期（10ms）调用一次,移动平均
fbMovingAvg_TiltSensorBottom(x := TiltSensorBottomAngle_mA,    // 输入原始值
            N := TiltSensorBottom_FilterWindow,  // 窗口大小
            rst := FALSE,       // 不复位
            y => TiltSensorBottomAngle_mA_Filter);     // 输出平均值
//计算角度
TiltSensorBottomAngle_Filter:=DINT_TO_LREAL(LREAL_TO_DINT(((TiltSensorBottomAngle_mA_Filter-12)*TiltSensorBottom_ScaleFactor+TiltSensorBottom_InitAngle)*100000))/100000;//滤波后
TiltSensorBottomAngle:=DINT_TO_LREAL(LREAL_TO_DINT(((TiltSensorBottomAngle_mA-12)*TiltSensorBottom_ScaleFactor+TiltSensorBottom_InitAngle)*100000))/100000;//未滤波，原始数据
//计算电机处由于倾斜导致的偏移量，单位毫米
//TileMotorOffset:=L_Center2Motor*2*TAN(TiltSensorAngle_degree*PI / 180);
//阈值触发
IF NormalGapMode THEN
	IF TiltSensorBottomAngle>TiltSensorBottom_GapThreshold THEN
		ErrorID:=1607;
		Error:=TRUE;
		ErrorDescription:='TiltSensorBottomAngle>TiltSensorBottom_Threshold';
		FB_PlcEmergencyStop();
		LED_Error:=TRUE;
	END_IF
END_IF
IF IDTaperMode THEN
	IF TiltSensorBottomAngle>TiltSensorBottom_IDTaperThreshold THEN
		ErrorID:=1608;
		Error:=TRUE;
		ErrorDescription:='TiltSensorBottomAngle>TiltSensorBottom_IDTaperThreshold';
		FB_PlcEmergencyStop();
		LED_Error:=TRUE;
	END_IF
END_IF
IF BLTaperMode THEN
	IF TiltSensorBottomAngle>TiltSensorBottom_BLTaperThreshold THEN
		ErrorID:=1609;
		Error:=TRUE;
		ErrorDescription:='TiltSensorBottomAngle>TiltSensorBottom_BLTaperThreshold';
		FB_PlcEmergencyStop();
		LED_Error:=TRUE;
	END_IF
END_IF
//角度与taper的比例
IF NormalGapMode THEN
	TaperAndTileBottomAngleScale:=0;
ELSIF IDTaperMode THEN
	TaperAndTileBottomAngleScale:=DINT_TO_LREAL(LREAL_TO_DINT((ATAN((UserMode.UserTaperPositionNew/2)/(2*UserMode.L_Center2Motor))*180/PI)*100000))/100000;;
ELSIF BLTaperMode THEN
	TaperAndTileBottomAngleScale:=DINT_TO_LREAL(LREAL_TO_DINT((ATAN((UserMode.BLUserTaperPositionNew/4)/(UserMode.L_HalfGirder))*180/PI)*100000))/100000;;
END_IF
//超出检测范围处理
IF TileSensorBottom_Underrange THEN
	ErrorID:=1610;
	Error:=TRUE;
	ErrorDescription:='TileSensorBottom_Underrange';
	//FB_PlcEmergencyStop();
	LED_Error:=TRUE;
ELSE
	ErrorID:=0;
	Error:=FALSE;
	ErrorDescription:='';
	LED_Error:=FALSE;
END_IF
IF TileSensorBottom_Overrange THEN
	ErrorID:=1611;
	Error:=TRUE;
	ErrorDescription:='TileSensorBottom_Overrange';
	//FB_PlcEmergencyStop();
	LED_Error:=TRUE;
ELSE
	ErrorID:=0;
	Error:=FALSE;
	ErrorDescription:='';
	LED_Error:=FALSE;
END_IF
IF TileSensorBottom_Error THEN
	ErrorID:=1612;
	Error:=TRUE;
	ErrorDescription:='TileSensorBottom_Error';
	//FB_PlcEmergencyStop();
	LED_Error:=TRUE;
ELSE
	ErrorID:=0;
	Error:=FALSE;
	ErrorDescription:='';
	LED_Error:=FALSE;
END_IF

END_PROGRAM

// ---- POUs/TiltSensor/FB_Simple_MovingAvg.TcPOU
FUNCTION_BLOCK FB_Simple_MovingAvg
VAR_INPUT
    x : LREAL;       // 输入值
    N : INT := 10;  // 平均点数
    rst : BOOL;     // 复位
END_VAR
VAR_OUTPUT
    y : LREAL;       // 平均值
END_VAR
VAR
    buf : ARRAY[0..999] OF LREAL;  // 固定50个点
    sum_x : LREAL;
    cnt : INT := 0;
    idx : INT := 0;
    n_actual : INT;
END_VAR

// 复位处理
IF rst THEN
    sum_x := 0.0;
    cnt := 0;
    idx := 0;
    y := 0.0;
    RETURN;
END_IF;

// 限制N在1-1000之间
n_actual := N;
IF n_actual < 1 THEN
    n_actual := 1;
ELSIF n_actual > 1000 THEN
    n_actual := 1000;
END_IF;

// 移动平均计算
IF cnt >= n_actual THEN
    // 缓冲区已满，减去最旧的值
    sum_x := sum_x - buf[idx];
ELSE
    // 缓冲区未满，只增加计数
    cnt := cnt + 1;
END_IF;

// 存入新值
buf[idx] := x;
sum_x := sum_x + x;

// 更新索引
idx := idx + 1;
IF idx >= n_actual THEN
    idx := 0;
END_IF;

// 计算平均值
IF cnt > 0 THEN
    y := sum_x / cnt;
ELSE
    y := 0.0;
END_IF;

END_FUNCTION_BLOCK

// ---- POUs/0.UserMode/UserMode.TcPOU
PROGRAM UserMode
VAR
(*GapMode*)
	UserGapPositionNew:LREAL:=20;//target
	UserGapVelocityNew:LREAL:=0.02;//target
	UserGapPositionDisplay:LREAL;//current
	UserGapVelocityDisplay:LREAL;//current
(*ID taper mode*)
	UserTaperPositionNew:LREAL:=0;//target
	UserTaperVelocityNew:LREAL:=0.02;//target
	UserTaperPositionDisplay:LREAL;//current
	UserTaperPositionDisplayBLSide:LREAL;//current BeamLine
	UserTaperPositionActual:LREAL;//current
	UserTaperVelocityDisplay:LREAL;//target
	UserGapPositionDisplay_FromLeftTop:LREAL;
	UserGapPositionDisplay_FromLeftBottom:LREAL;
		//
	UserRightGapPositionNew:LREAL;
	UserRightGapVelocityNew:LREAL;
	UserRightGapPositionDisplay:LREAL;
	UserRightGapVelocityDisplay:LREAL;
	UserRightGapPositionDisplay_FromRightTop:LREAL;
	UserRightGapPositionDisplay_FromRightBottom:LREAL;
(*BL taper mode*)
	BLUserTaperPositionNew:LREAL:=0;//target
	BLUserTaperVelocityNew:LREAL:=0.02;//target
	BLUserTaperPositionDisplay:LREAL;//current
	//BLUserTaperPositionDisplayBLSide:LREAL;//current BeamLine
	BLUserTaperPositionActual:LREAL;//current
	BLUserTaperVelocityDisplay:LREAL;//target
	BLUserGapPositionDisplay_FromLeftTop:LREAL;
	BLUserGapPositionDisplay_FromLeftBottom:LREAL;
	//
	BLUserLeftGapPositionNew:LREAL;
	BLUserLeftGapVelocityNew:LREAL;
	BLUserLeftGapPositionDisplay:LREAL;
	BLUserLeftGapVelocityDisplay:LREAL;
	BLUserLeftGapPositionDisplay_FromLeftTop:LREAL;
	BLUserLeftGapPositionDisplay_FromLeftBottom:LREAL;
	BLUserRightGapPositionNew:LREAL;
	BLUserRightGapVelocityNew:LREAL;
	BLUserRightGapPositionDisplay:LREAL;
	BLUserRightGapVelocityDisplay:LREAL;
	BLUserRightGapPositionDisplay_FromRightTop:LREAL;
	BLUserRightGapPositionDisplay_FromRightBottom:LREAL;

	(**)
	btn_UserGapMove:BOOL;
	btn_UserGapStop:BOOL;
	(*Var*)
	fb_ton1:TON;
	fb_ton2:TON;
	fb_ton3:TON;
	(*Status*)
	State:DINT;
	Busy:BOOL;
	InitPowerDone:BOOL;
	InitCompensationDatasDone:BOOL;
	(*FB*)
	m_state: DINT;
	n_state: DINT;
	s_state: DINT;
	(*¼ì²âµ½ÏÞÎ»£¬»Ö¸´Move×´Ì¬*)
	FTrig_ReachLS: F_TRIG;
	FTrig_btn_GapMove: F_TRIG;
	GapOutRange: BOOL;
	(*PowerOff*)
	d_state: DINT;
	i: INT;
	j: INT;
	k: INT;
	moni_State:DINT;
	TargetPosLessThanCurrentPos:BOOL;
	TargetLTPosLessThanCurrentLTPos:BOOL;
	TargetRTPosLessThanCurrentRTPos:BOOL;
	TargetLBPosLessThanCurrentLBPos:BOOL;
	TargetRBPosLessThanCurrentRBPos:BOOL;
	PositiveMoving:BOOL;
	HysteresisMoving:BOOL;
	NoneHysteresisMoving:BOOL;
	(*Spectroscopy scanning Mode*)
	IsSSMotionMode:BOOL;
	RegularMotionMode:BOOL;
	SSMotionMode:BOOL;
	SS_StepSize:LREAL:=0.001;
	SS_StepNumber:INT:=10;
	SS_StepVelocity:LREAL:=1;
	SS_Move:BOOL;
	SS_Stop:BOOL;
	SS_MoveState:DINT;
	SS_StopState:DINT;
	SS_currentStep:DINT:=0;
	SS_StepSystemTime_Begin:ARRAY[0..100] OF ULINT;
	SS_StepSystemTime_End:ARRAY[0..100] OF ULINT;
	SS_StepCountTime:ARRAY[0..100] OF ULINT;
	SS_TimeCountBegin:BOOL;
	m: INT;
	SS_TON: TON;
	StepEachTime:TIME;
	StepEachTime_ms:INT:=1000;//ms
	SS_OTSTRUCT :OTSTRUCT ;
	SS_StartPositionDisplay:LREAL;
	RTRG_SS_StartPositionDisplay:R_TRIG;
	SS_InitStartPositionDone:BOOL;

	//
	min_SS_StepSize	: LREAL:=0;
	max_SS_StepSize	: LREAL:=200;
	inRange_SS_StepSize	: BOOL;
	//
	min_SS_StepNumber	: INT:=1;
	max_SS_StepNumber	: INT:=1000;
	inRange_SS_StepNumber	: BOOL;
	//
	min_SS_StepVelocity:LREAL:=0;
	max_SS_StepVelocity:LREAL:=1;
	inRange_SS_StepVelocity:BOOL;
	//
	min_StepEachTime_ms:INT:=100;
	max_StepEachTime_ms:INT:=10000;
	inRange_StepEachTime_ms:BOOL;
	l: INT;
	Threshold_UserTopPos_PLC: LREAL;
	Threshold_UserTopVelo_PLC: LREAL;
	Threshold_UserBottomPos_PLC: LREAL;
	Threshold_UserBottomVelo_PLC: LREAL;
	Threshold_UserLeftPos_PLC: LREAL;
	Threshold_UserLeftVelo_PLC: LREAL;
	Threshold_UserRightPos_PLC: LREAL;
	Threshold_UserRightVelo_PLC: LREAL;
	testa: BOOL;
	testb: BOOL;
	//Taper parameters
	Threshold_GapChangeFlag: LREAL:=0.001;
	Threshold_TaperChangeFlag: LREAL:=0.005;
	TaperAndGapSafetyfactor: LREAL:=1;
	TaperAndGapSafetyScale:LREAL:=0.41;//IAU=0.409,IVU=0.32,CPMU=0.328,IAMW=0.42
	TaperAndGapSafetyMinGapMargin:LREAL:=0.2;
	IDTaperAndBLTaperScale:LREAL:=0.548;//HU 
	//HEPSIDTaperAndBLTaperScale:LREAL:=0.55;
	//
	//Global Chain protection-MPS
	Global_ChainProtection_MPS_StorageRingReady:BOOL;
	Global_ChainProtection_MPS_On: BOOL;
	Global_ChainProtection_MPS_MaxGapValue: LREAL;
	Global_ChainProtection_MPS_MoveVelocity: LREAL;
	Global_ChainProtection_MPS_Done: BOOL;
	//Global_ChainProtection_Error: BOOL;
	//Global_ChainProtection_ErrorID: INT;
	//Global_ChainProtection_ErrorDescription: STRING;
	Global_ChainProtection_MPS_ManualOperation:BOOL:=TRUE;
	Global_ChainProtection_MPS_FTRIG:F_TRIG;
	Global_ChainProtection_MPS_FTRIG_Manul:F_TRIG;
	Global_ChainProtection_MPS_TON:TON;
	Global_ChainProtection_MPS_Triggered:BOOL;
	Global_ChainProtection_MPS_In:BOOL;
	Global_ChainProtection_MPS_In1 AT%I* :BOOL;//下降沿表示触发,EL1008
	Global_ChainProtection_MPS_In2 AT%I* :BOOL;
	Global_ChainProtection_MPS_State:DINT;
	Global_ChainProtection_MPS_Out1 AT%Q* :BOOL;//上升沿标识到达最大间隙，连锁保护成功,EL2624
	Global_ChainProtection_MPS_Out2 AT%Q* :BOOL;
	Global_ChainProtection_MPS_TON_Stop2Move:TON;
	Global_ChainProtection_MPS_TON_Stop2Move_InTaperMode:TON;
	Global_ChainProtection_MPS_TON_Power2Move:TON;
	//Global Chain protection-EPS
	Global_ChainProtection_EPS_BeamLineReady:BOOL;
	Global_ChainProtection_EPS_On: BOOL;
	Global_ChainProtection_EPS_MaxGapValue: LREAL;
	Global_ChainProtection_EPS_MoveVelocity: LREAL;
	Global_ChainProtection_EPS_Done: BOOL;
	//Global_ChainProtection_Error: BOOL;
	//Global_ChainProtection_ErrorID: INT;
	//Global_ChainProtection_ErrorDescription: STRING;
	Global_ChainProtection_EPS_ManualOperation:BOOL:=TRUE;
	Global_ChainProtection_EPS_FTRIG:F_TRIG;
	Global_ChainProtection_EPS_FTRIG_Manul:F_TRIG;
	Global_ChainProtection_EPS_TON:TON;
	Global_ChainProtection_EPS_Triggered:BOOL;
	Global_ChainProtection_EPS_In:BOOL;
	Global_ChainProtection_EPS_In1 AT%I* :BOOL;//下降沿表示触发,EL1124
	Global_ChainProtection_EPS_In2 AT%I* :BOOL;
	Global_ChainProtection_EPS_State:DINT;
	Global_ChainProtection_EPS_Out1 AT%Q* :BOOL;//上升沿标识到达最大间隙，连锁保护成功,EL2124
	Global_ChainProtection_EPS_Out2 AT%Q* :BOOL;
	Global_ChainProtection_EPS_TON_Stop2Move:TON;
	Global_ChainProtection_EPS_TON_Stop2Move_InTaperMode:TON;
	Global_ChainProtection_EPS_TON_Power2Move:TON;
	//
	//Cryogenic Chain protection
	Cryogenic_ChainProtection_On: BOOL;
	Cryogenic_ChainProtection_MaxGapValue: LREAL;
	Cryogenic_ChainProtection_MoveVelocity: LREAL;
	Cryogenic_ChainProtection_Done: BOOL;
	//Cryogenic_ChainProtection_Error: BOOL;
	//Cryogenic_ChainProtection_ErrorID: INT;
	//Cryogenic_ChainProtection_ErrorDescription: STRING;
	Cryogenic_ChainProtection_ManualOperation:BOOL:=TRUE;
	Cryogenic_ChainProtection_FTRIG:F_TRIG;
	Cryogenic_ChainProtection_FTRIG_Manul:F_TRIG;
	Cryogenic_ChainProtection_TON:TON;
	Cryogenic_ChainProtection_Triggered:BOOL;
	Cryogenic_ChainProtection_In:BOOL;
	Cryogenic_ChainProtection_State:DINT;
	Cryogenic_ChainProtection_Out1 AT%Q* :BOOL;//上升沿标识到达最大间隙，连锁保护成功
	Cryogenic_ChainProtection_TON_Stop2Move:TON;
	Cryogenic_ChainProtection_TON_Stop2Move_InTaperMode:TON;
	Cryogenic_ChainProtection_TON_Power2Move:TON;
	test11:INT:=1;
	IsTest11OrNot:BOOL;
	tesetBegin: BOOL;
	Threshold_motorsTargetPosCalculate: LREAL;
	SS_Stop2: BOOL;
	//
	LeftTopLinPositionNewTemp: LREAL;
	RightTopLinPositionNewTemp: LREAL;
	LeftBottomLinPositionNewTemp: LREAL;
	RightBottomLinPositionNewTemp: LREAL;
	
	
	//OneKeyToMaxGap
	btn_OneKeyToMaxGap:BOOL;
	OneKeyToMaxGap_RTRIG:R_TRIG;
	OneKeyToMaxGap_TON:TON;
	OneKeyToMaxGap_Triggered:BOOL;
	OneKeyToMaxGap_State:DINT;
	OneKeyToMaxGap_TON_Stop2Move:TON;
	OneKeyToMaxGap_TON_Stop2Move_InTaperMode:TON;
	OneKeyToMaxGap_TON_Power2Move:TON;
	OneKeyToMaxGap_Done:BOOL;
	FTrig_ReachLSa: F_TRIG;
	Unreach_LS_Fara: BOOL;
	Unreach_LS_Neara: BOOL;
	btn_UserGapStopa: BOOL;
	
	//OneKeyToMTaperZero
	btn_OneKeyToTaperZero:BOOL;
	OneKeyToTaperZero_RTRIG:R_TRIG;
	OneKeyToTaperZero_TON:TON;
	OneKeyToTaperZero_Triggered:BOOL;
	OneKeyToTaperZero_State:DINT;
	OneKeyToTaperZero_Done:BOOL;
	OneKeyToTaperZero_Delay:TON;
	//BLTaper
	CurrentTaperInit: LREAL;
	L_HalfGirder:LREAL:=2500;
	L_Center2Motor:LREAL:=1375;
	
	trig_TaperOrNot: R_TRIG;
	trig_BLTaperOrNot: R_TRIG;
END_VAR

IF NOT PositionBiasDone THEN
	RETURN;
END_IF
IF NOT loadParametersDone THEN
	RETURN;
END_IF
(*btn_Power On/Off*)
IF btn_Power AND NOT st_Power THEN
	btn_PowerOn:=TRUE;
	btn_Power:=FALSE;
END_IF
IF btn_Power AND st_Power THEN
	btn_PowerOff:=TRUE;
	btn_Power:=FALSE;
END_IF
IF btn_PowerOn THEN
	A_PowerOn();
END_IF
IF btn_PowerOff THEN
	A_PowerOff();
END_IF

(*检查couple状态，不允许couple*)
A_CheckCoupleStatus();

(*监控四轴位置速度等*)
A_MonitoringAllAxis();

(*目标位置和速度保护*)
A_CheckMotorsPos();

(*补偿数据处理*)
A_InitCompensationData();

(*常规磁间隙开合*)
IF RegularMotionMode AND NOT SSMotionMode THEN
	A_RegularMotion();
END_IF

(*Spectroscopy scanning Mode*)
IF IsSSMotionMode THEN
	SSMotionMode:=TRUE;
	RegularMotionMode:=FALSE;
ELSE
	SSMotionMode:=FALSE;
	RegularMotionMode:=TRUE;
END_IF
IF	SSMotionMode AND NOT RegularMotionMode THEN
	A_SpectroscopyScanningMotion();
END_IF


(*GlobalChainProtection*)
A_GlobalChainProtection_MPS();
A_GlobalChainProtection_EPS();

(*CryogenicChainProtection*)
A_CryogenicChainProtection();

(*A_OneKeyToMaxGap*)
A_OneKeyToMaxGap();

(*A_OneKeyToTaperZero*)
A_OneKeyToTaperZero();

(*A_TaperParametersInit*)
A_TaperParametersInit();

ACTION A_CheckCoupleStatus:
IF NOT btn_PowerOff THEN
	IF st_Power=1 AND st_Couple<>0THEN
		Error:=TRUE;
		ErrorID:=501;
		LeftTopLinMoveIndicator:=0;
		RightTopLinMoveIndicator:=0;
		LeftBottomLinMoveIndicator:=0;
		RightBottomLinMoveIndicator:=0;
		FB_PlcEmergencyStop();
		LED_Error:=TRUE;
		ErrorDescription:='couple stutas error';
	END_IF
END_IF
END_ACTION

ACTION A_CheckMotorsPos:
//
//目标位置速度超出阈值判断
//
//gap posiion
IF UserGapPositionNew<min_UserGapPositionNew OR UserGapPositionNew>max_UserGapPositionNew THEN
	inRange_UserGapPositionNew:=FALSE;
END_IF
IF UserGapPositionNew>=min_UserGapPositionNew AND UserGapPositionNew<=max_UserGapPositionNew THEN
	inRange_UserGapPositionNew:=TRUE;
END_IF
//gap velocity
IF UserGapVelocityNew<min_UserGapVelocityNew OR UserGapVelocityNew>max_UserGapVelocityNew THEN
	inRange_UserGapVelocityNew:=FALSE;
END_IF
IF UserGapVelocityNew>=min_UserGapVelocityNew AND UserGapVelocityNew<=max_UserGapVelocityNew THEN
	inRange_UserGapVelocityNew:=TRUE;
END_IF
//IDtaper position
IF UserTaperPositionNew<min_UserTaperPositionNew OR UserTaperPositionNew>max_UserTaperPositionNew THEN
	inRange_UserTaperPositionNew:=FALSE;
END_IF
IF UserTaperPositionNew>=min_UserTaperPositionNew AND UserTaperPositionNew<=max_UserTaperPositionNew THEN
	inRange_UserTaperPositionNew:=TRUE;
END_IF
//IDtaper velocity
IF UserTaperVelocityNew<min_UserTaperVelocityNew OR UserTaperVelocityNew>max_UserTaperVelocityNew THEN
	inRange_UserTaperVelocityNew:=FALSE;
END_IF
IF UserTaperVelocityNew>=min_UserTaperVelocityNew AND UserTaperVelocityNew<=max_UserTaperVelocityNew THEN
	inRange_UserTaperVelocityNew:=TRUE;
END_IF
//BLtaper position
IF BLUserTaperPositionNew<min_BLUserTaperPositionNew OR BLUserTaperPositionNew>max_BLUserTaperPositionNew THEN
	inRange_BLUserTaperPositionNew:=FALSE;
END_IF
IF BLUserTaperPositionNew>=min_BLUserTaperPositionNew AND BLUserTaperPositionNew<=max_BLUserTaperPositionNew THEN
	inRange_BLUserTaperPositionNew:=TRUE;
END_IF
//BLtaper velocity
IF BLUserTaperVelocityNew<min_BLUserTaperVelocityNew OR BLUserTaperVelocityNew>max_BLUserTaperVelocityNew THEN
	inRange_BLUserTaperVelocityNew:=FALSE;
END_IF
IF BLUserTaperVelocityNew>=min_BLUserTaperVelocityNew AND BLUserTaperVelocityNew<=max_BLUserTaperVelocityNew THEN
	inRange_BLUserTaperVelocityNew:=TRUE;
END_IF
//SS Mode
IF SS_StepSize<min_SS_StepSize OR SS_StepSize>max_SS_StepSize THEN
	inRange_SS_StepSize:=FALSE;
END_IF
IF SS_StepSize>=min_SS_StepSize AND SS_StepSize<=max_SS_StepSize THEN
	inRange_SS_StepSize:=TRUE;
END_IF
IF SS_StepNumber<min_SS_StepNumber OR SS_StepNumber>max_SS_StepNumber THEN
	inRange_SS_StepNumber:=FALSE;
END_IF
IF SS_StepNumber>=min_SS_StepNumber AND SS_StepNumber<=max_SS_StepNumber THEN
	inRange_SS_StepNumber:=TRUE;
END_IF
IF SS_StepVelocity<min_SS_StepVelocity OR SS_StepVelocity>max_SS_StepVelocity THEN
	inRange_SS_StepVelocity:=FALSE;
END_IF
IF SS_StepVelocity>=min_SS_StepVelocity AND SS_StepVelocity<=max_SS_StepVelocity THEN
	inRange_SS_StepVelocity:=TRUE;
END_IF
IF StepEachTime_ms<min_StepEachTime_ms OR StepEachTime_ms>max_StepEachTime_ms THEN
	inRange_StepEachTime_ms:=FALSE;
END_IF
IF StepEachTime_ms>=min_StepEachTime_ms AND StepEachTime_ms<=max_StepEachTime_ms THEN
	inRange_StepEachTime_ms:=TRUE;
END_IF


//
//输入速度和位置保护
//
IF btn_UserGapMove  AND NOT SSMotionMode AND RegularMotionMode THEN
	IF NOT inRange_UserGapPositionNew THEN
		btn_UserGapStop:=TRUE;
		btn_UserGapMove:=FALSE;
		Error:=TRUE;
		ErrorId:=801;
		ErrorDescription:='target Gap position out of range,please check';
		RETURN;
	ELSE
		//btn_UserGapStop:=FALSE;
		Error:=FALSE;
		ErrorId:=0;
		ErrorDescription:='';	
	END_IF
	IF NOT inRange_UserGapVelocityNew THEN
		btn_UserGapStop:=TRUE;
		btn_UserGapMove:=FALSE;
		Error:=TRUE;
		ErrorId:=802;
		ErrorDescription:='target Gap velocity out of range,please check';
		RETURN;
	ELSE
		//btn_UserGapStop:=FALSE;
		Error:=FALSE;
		ErrorId:=0;
		ErrorDescription:='';
	END_IF
	IF NOT inRange_UserTaperPositionNew THEN
		btn_UserGapStop:=TRUE;
		btn_UserGapMove:=FALSE;
		Error:=TRUE;
		ErrorId:=803;
		ErrorDescription:='target Taper Position out of range,please check';
		RETURN;
	ELSE
		//btn_UserGapStop:=FALSE;
		Error:=FALSE;
		ErrorId:=0;
		ErrorDescription:='';
	END_IF
	IF NOT inRange_UserTaperVelocityNew THEN
		btn_UserGapStop:=TRUE;
		btn_UserGapMove:=FALSE;
		Error:=TRUE;
		ErrorId:=804;
		ErrorDescription:='target Taper velocity out of range,please check';
		RETURN;
	ELSE
		//btn_UserGapStop:=FALSE;
		Error:=FALSE;
		ErrorId:=0;
		ErrorDescription:='';
	END_IF
	IF NOT inRange_BLUserTaperPositionNew THEN
		btn_UserGapStop:=TRUE;
		btn_UserGapMove:=FALSE;
		Error:=TRUE;
		ErrorId:=805;
		ErrorDescription:='target BLTaper Position out of range,please check';
		RETURN;
	ELSE
		//btn_UserGapStop:=FALSE;
		Error:=FALSE;
		ErrorId:=0;
		ErrorDescription:='';
	END_IF
	IF NOT inRange_BLUserTaperVelocityNew THEN
		btn_UserGapStop:=TRUE;
		btn_UserGapMove:=FALSE;
		Error:=TRUE;
		ErrorId:=806;
		ErrorDescription:='target BLTaper velocity out of range,please check';
		RETURN;
	ELSE
		//btn_UserGapStop:=FALSE;
		Error:=FALSE;
		ErrorId:=0;
		ErrorDescription:='';
	END_IF
END_IF

//
//运动过程中，监控目标位置速度
//
IF moveStatusAnyAxis THEN
	IF NOT inRange_UserGapPositionNew THEN
		btn_UserGapStop:=TRUE;
		Error:=TRUE;
		ErrorId:=807;
		ErrorDescription:='target Gap position out of range in moving process!';
		FB_PlcEmergencyStop();
	END_IF
	IF NOT inRange_UserGapVelocityNew THEN
		btn_UserGapStop:=TRUE;
		Error:=TRUE;
		ErrorId:=808;
		ErrorDescription:='target Gap velocity out of range in moving process!';
		FB_PlcEmergencyStop();
	END_IF
	IF NOT inRange_UserTaperPositionNew THEN
		btn_UserGapStop:=TRUE;
		Error:=TRUE;
		ErrorId:=809;
		ErrorDescription:='target Taper Position out of range in moving process!';
		FB_PlcEmergencyStop();
	END_IF
	IF NOT inRange_UserTaperVelocityNew THEN
		btn_UserGapStop:=TRUE;
		Error:=TRUE;
		ErrorId:=810;
		ErrorDescription:='target Taper velocity out of range in moving process!';
		FB_PlcEmergencyStop();
	END_IF
	IF NOT inRange_BLUserTaperPositionNew THEN
		btn_UserGapStop:=TRUE;
		Error:=TRUE;
		ErrorId:=811;
		ErrorDescription:='target BLTaper Position out of range in moving process!';
		FB_PlcEmergencyStop();
	END_IF
	IF NOT inRange_BLUserTaperVelocityNew THEN
		btn_UserGapStop:=TRUE;
		Error:=TRUE;
		ErrorId:=812;
		ErrorDescription:='target BLTaper velocity out of range in moving process!';
		FB_PlcEmergencyStop();
	END_IF
END_IF
//
//运动过程中，监控每一个轴的目标位置，目标位置若超出阈值，Emergency
//
IF moveStatusAnyAxis THEN
	IF NormalGapMode THEN
		IF LeftTopLinPositionNew<min_UserLEProtectionGapPosition/2 OR LeftTopLinPositionNew>max_UserLEProtectionGapPosition/2 THEN
			btn_UserGapStop:=TRUE;
			Error:=TRUE;
			ErrorId:=809;
			ErrorDescription:='target LeftTop position out of range in moving process!';
			FB_PlcEmergencyStop();
		END_IF
		IF RightTopLinPositionNew<min_UserLEProtectionGapPosition/2 OR RightTopLinPositionNew>max_UserLEProtectionGapPosition/2 THEN
			btn_UserGapStop:=TRUE;
			Error:=TRUE;
			ErrorId:=810;
			ErrorDescription:='target RightTop velocity out of range in moving process!';
			FB_PlcEmergencyStop();
		END_IF
		IF LeftBottomLinPositionNew<min_UserLEProtectionGapPosition/2 OR LeftBottomLinPositionNew>max_UserLEProtectionGapPosition/2 THEN
			btn_UserGapStop:=TRUE;
			Error:=TRUE;
			ErrorId:=812;
			ErrorDescription:='target LeftBottom Position out of range in moving process!';
			FB_PlcEmergencyStop();
		END_IF
		IF RightBottomLinPositionNew<min_UserLEProtectionGapPosition/2 OR RightBottomLinPositionNew>max_UserLEProtectionGapPosition/2 THEN
			btn_UserGapStop:=TRUE;
			Error:=TRUE;
			ErrorId:=813;
			ErrorDescription:='target RightBottom Position out of range in moving process!';
			FB_PlcEmergencyStop();
		END_IF
	ELSE//Taper状态的保护
		;//Taper状态下，不用监控四轴位置，只需要监控目标Taper位置。在上面已经保护
	END_IF
END_IF
END_ACTION

ACTION A_CryogenicChainProtection:
//总开关
IF NOT Cryogenic_ChainProtection_On THEN
	RETURN;
END_IF
IF NOT MAIN.CryogenicCompensationOn THEN
	RETURN;
END_IF
//判断插入件状态，是否就位
//IF NOT IDControlReady THEN
//	Cryogenic_ChainProtection_Done:=FALSE;
//	Error:= TRUE;
//	ErrorID:=1501;
//	ErrorDescription:='ID NOT READY!';
//	RETURN;
//END_IF

//
//全局连锁保护程序开始
//
//0.检测温度变化超出正常范围，或者手动触发，触发低温联锁保护
//1.判断电机是否在开启状态,没有就打开电源
//2.判断是否在Moving状态,若有就Stop
//3.将磁间隙打开到至最大阈值
//4.到位后给出反馈，且安全PLC触发
//IF MAIN.temperatureStatus=3 THEN //=2低温,超出低温阈值就触发保护
//	Cryogenic_ChainProtection_Triggered:=TRUE;
//END_IF
Cryogenic_ChainProtection_FTRIG(CLK:=MAIN.InCryogenicOrNot);
IF Cryogenic_ChainProtection_FTRIG.Q THEN
	Cryogenic_ChainProtection_Triggered:=TRUE;
END_IF
Cryogenic_ChainProtection_FTRIG_Manul(CLK:=Cryogenic_ChainProtection_ManualOperation);
IF Cryogenic_ChainProtection_FTRIG_Manul.Q THEN
	Cryogenic_ChainProtection_Triggered:=TRUE;
END_IF
IF Cryogenic_ChainProtection_Triggered THEN
	//判断当前间隙，如果比Cryogenic_ChainProtection_MaxGapValue大，则不动作，只报警，且安全PLC触发
	IF UserGapPositionDisplay - Cryogenic_ChainProtection_MaxGapValue >=0.001THEN
		Cryogenic_ChainProtection_Done:=TRUE;
		Plc_EmergencyStop:=FALSE;
		Error:= TRUE;
		ErrorID:= 1502;
		ErrorDescription:='Cryogenic Abnormal !';
		RETURN;
	END_IF
	CASE Cryogenic_ChainProtection_State OF
		0://1.判断电机是否在开启状态,没有就打开电源
			IF st_Power=1 THEN
				Cryogenic_ChainProtection_State:=1;
			ELSE
				btn_PowerOn:=TRUE;
				IF btn_PowerOn THEN
					A_PowerOn();
				END_IF
			END_IF
		1://1.判断是否在谱学扫描模式，如果是，则切换回正常运动模式
			IF IsSSMotionMode THEN
				SS_Stop:=TRUE;
				IsSSMotionMode:=FALSE;
			END_IF
			Cryogenic_ChainProtection_State:=2;
		2://判断是否在taper，如果在taper,则判断是否在运动，如果是，则停止运动,0.5sh后，转入下一步
			IF TaperOrNot THEN
				IF moveStatusLeftTop OR moveStatusRightTop OR moveStatusLeftBottom OR moveStatusRightBottom THEN
					btn_UserGapStop:=TRUE;
				ELSE
					Cryogenic_ChainProtection_TON_Stop2Move_InTaperMode(PT:=T#0.5S);
					Cryogenic_ChainProtection_TON_Stop2Move_InTaperMode.IN:=TRUE;
					IF Cryogenic_ChainProtection_TON_Stop2Move_InTaperMode.Q THEN
						TaperOrNot:=FALSE;//关闭taper模式
						Cryogenic_ChainProtection_State:=3;
					END_IF
				END_IF
			ELSE
				Cryogenic_ChainProtection_State:=3;
			END_IF
		3://3.判断是否在Moving状态,若有就Stop.Taper模式已处理完，此处开始走正常GAP开合逻辑
			IF moveStatusLeftTop OR moveStatusRightTop OR moveStatusLeftBottom OR moveStatusRightBottom THEN
				btn_UserGapStop:=TRUE;
			ELSE
				Cryogenic_ChainProtection_TON_Stop2Move(PT:=T#0.5S);
				Cryogenic_ChainProtection_TON_Stop2Move.IN:=TRUE;
				IF Cryogenic_ChainProtection_TON_Stop2Move.Q THEN
					Cryogenic_ChainProtection_State:=4;
				END_IF
			END_IF
		4://4.将磁间隙打开到至最大阈值
			Cryogenic_ChainProtection_TON(PT:=INT_TO_TIME(LREAL_TO_INT(Cryogenic_ChainProtection_MaxGapValue/Cryogenic_ChainProtection_MoveVelocity+30))*1000);
			Cryogenic_ChainProtection_TON.IN:=TRUE;
			Cryogenic_ChainProtection_TON_Power2Move(PT:=T#0.1S);
			Cryogenic_ChainProtection_TON_Power2Move.IN:=TRUE;
			UserGapPositionNew:=Cryogenic_ChainProtection_MaxGapValue;
			UserGapVelocityNew:=Cryogenic_ChainProtection_MoveVelocity;
			btn_UserGapMove:=TRUE;
			IF Cryogenic_ChainProtection_TON_Power2Move.Q THEN
				IF FB_MOVE.BCGapDone THEN
					Cryogenic_ChainProtection_State:=88;
				END_IF
			END_IF
			IF Cryogenic_ChainProtection_TON.Q THEN//如果150s后，还没有运动到指定gap，则报错
				Cryogenic_ChainProtection_State:=-100;
			END_IF
		88://4.到位后给出反馈，且安全PLC触发
			Cryogenic_ChainProtection_Done:=TRUE;
			Plc_EmergencyStop:=FALSE;		
			Error:=TRUE;
			ErrorID:=1503;
			ErrorDescription:='Cryogenic_ChainProtection Triggered';
		-100:
			Cryogenic_ChainProtection_Done:=FALSE;
			Error:=TRUE;
			ErrorID:=1504;
			ErrorDescription:='NOT MOVING TO MAXGAP';
	END_CASE
END_IF

//监控是否同时是低温模式，且温度传感器检测到的是低温+10℃（避开低温联锁保护，联锁保护要求在低温阈值时拉开磁间隙）
IF MAIN.temperatureStatus<>0 AND MAIN.temperature_average > MAIN.CryogenicTemperatureThreshold +10 THEN//在低温+10℃
	IF MAIN.HasTemperatureSensorOrNot AND MAIN.CryogenicCompensationOn THEN
			Error:=TRUE;
			ErrorID:=1505;
			Plc_EmergencyStop:=FALSE;
			ErrorDescription:='CryogenicCompensationOn AND Room temperatureStatus';
	END_IF
END_IF
END_ACTION

ACTION A_GlobalChainProtection_EPS:
//硬线输入定义
Global_ChainProtection_EPS_In:=Global_ChainProtection_EPS_In1 AND Global_ChainProtection_EPS_In2;
//硬线输出定义
Global_ChainProtection_EPS_Out1:=Global_ChainProtection_EPS_Done;
Global_ChainProtection_EPS_Out2:=Global_ChainProtection_EPS_Done;
//总开关
IF NOT Global_ChainProtection_EPS_On THEN
	RETURN;
END_IF
//判断插入件状态，是否就位
//IF NOT IDControlReady THEN
//	Global_ChainProtection_EPS_Done:=FALSE;
//	Error:= TRUE;
//	ErrorID:= 1501;
//	ErrorDescription:='ID NOT READY!';
//	RETURN;
//END_IF
//判断储存环是否给出就位信号，暂时由参数表给出TRUE，最终将由IOC接受PV
IF 	NOT Global_ChainProtection_EPS_BeamLineReady THEN
	Global_ChainProtection_EPS_Done:=FALSE;
	Error:= TRUE;
	ErrorID:= 1503;
	ErrorDescription:='Global_ChainProtection_EPS_BeamLineReady NOT Ready';
	RETURN;
END_IF
//
//全局连锁保护程序开始
//
//0.检测到下降沿，触发
//1.判断电机是否在开启状态,没有就打开电源
//2.判断是否在Moving状态,若有就Stop
//3.将磁间隙打开到至最大阈值
//4.到位后给出反馈，且安全PLC触发
Global_ChainProtection_EPS_FTRIG(CLK:=Global_ChainProtection_EPS_In);
IF Global_ChainProtection_EPS_FTRIG.Q THEN
	Global_ChainProtection_EPS_Triggered:=TRUE;
END_IF
Global_ChainProtection_EPS_FTRIG_Manul(CLK:=Global_ChainProtection_EPS_ManualOperation);
IF Global_ChainProtection_EPS_FTRIG_Manul.Q THEN
	Global_ChainProtection_EPS_Triggered:=TRUE;
END_IF
IF Global_ChainProtection_EPS_Triggered THEN
	CASE Global_ChainProtection_EPS_State OF
		0://1.判断电机是否在开启状态,没有就打开电源
			IF st_Power=1 THEN
				Global_ChainProtection_EPS_State:=1;
			ELSE
				btn_PowerOn:=TRUE;
				IF btn_PowerOn THEN
					A_PowerOn();
				END_IF
			END_IF
		1://1.判断是否在谱学扫描模式，如果是，则切换回正常运动模式
			IF IsSSMotionMode THEN
				SS_Stop:=TRUE;
				IsSSMotionMode:=FALSE;
			END_IF
			Global_ChainProtection_EPS_State:=2;
		2://判断是否在taper，如果在taper,则判断是否在运动，如果是，则停止运动,0.5sh后，转入下一步
			IF TaperOrNot THEN
				IF moveStatusLeftTop OR moveStatusRightTop OR moveStatusLeftBottom OR moveStatusRightBottom THEN
					btn_UserGapStop:=TRUE;
				ELSE
					Global_ChainProtection_EPS_TON_Stop2Move_InTaperMode(PT:=T#0.5S);
					Global_ChainProtection_EPS_TON_Stop2Move_InTaperMode.IN:=TRUE;
					IF Global_ChainProtection_EPS_TON_Stop2Move_InTaperMode.Q THEN
						TaperOrNot:=FALSE;//关闭taper模式
						Global_ChainProtection_EPS_State:=3;
					END_IF
				END_IF
			ELSE
				Global_ChainProtection_EPS_State:=3;
			END_IF
		3://3.判断是否在Moving状态,若有就Stop.Taper模式已处理完，此处开始走正常GAP开合逻辑
			IF moveStatusLeftTop OR moveStatusRightTop OR moveStatusLeftBottom OR moveStatusRightBottom THEN
				btn_UserGapStop:=TRUE;
			ELSE
				Global_ChainProtection_EPS_TON_Stop2Move(PT:=T#0.5S);
				Global_ChainProtection_EPS_TON_Stop2Move.IN:=TRUE;
				IF Global_ChainProtection_EPS_TON_Stop2Move.Q THEN
					Global_ChainProtection_EPS_State:=4;
				END_IF
			END_IF
		4://当前磁间隙如何和最大磁间隙差别不大，不超过0.1，则直接保护
			IF ABS(UserGapPositionDisplay-Global_ChainProtection_EPS_MaxGapValue)<=0.1 THEN
				Global_ChainProtection_EPS_Done:=TRUE;
				Plc_EmergencyStop:=FALSE;	
				Error:=TRUE;
				ErrorID:=1506;
				ErrorDescription:='EPS Triggered,but ABS(GapPositionDisplay-EPS_MaxGapValue)<=0.1 ';	
			ELSE
				Global_ChainProtection_EPS_State:=5;
			END_IF
		5://5.将磁间隙打开到至最大阈值
			Global_ChainProtection_EPS_TON(PT:=INT_TO_TIME(LREAL_TO_INT(Global_ChainProtection_EPS_MaxGapValue/Global_ChainProtection_EPS_MoveVelocity+30))*1000);
			Global_ChainProtection_EPS_TON.IN:=TRUE;
			Global_ChainProtection_EPS_TON_Power2Move(PT:=T#0.1S);
			Global_ChainProtection_EPS_TON_Power2Move.IN:=TRUE;
			UserGapPositionNew:=Global_ChainProtection_EPS_MaxGapValue;
			UserGapVelocityNew:=Global_ChainProtection_EPS_MoveVelocity;
			btn_UserGapMove:=TRUE;
			IF Global_ChainProtection_EPS_TON_Power2Move.Q THEN
				IF FB_MOVE.BCGapDone THEN
					Global_ChainProtection_EPS_State:=88;
				END_IF
			END_IF
			IF Global_ChainProtection_EPS_TON.Q THEN//如果150s后，还没有运动到指定gap，则报错
				Global_ChainProtection_EPS_State:=-100;
			END_IF
		88://6.到位后给出反馈，且安全PLC触发
			Global_ChainProtection_EPS_Done:=TRUE;
			Plc_EmergencyStop:=FALSE;	
			Error:=TRUE;
			ErrorID:=1504;
			ErrorDescription:='Global_ChainProtection_EPS Triggered ';	
		-100:
			Global_ChainProtection_EPS_Done:=FALSE;
			Error:=TRUE;
			ErrorID:=1505;
			ErrorDescription:='NOT MOVING TO MAXGAP';
	END_CASE
END_IF
END_ACTION

ACTION A_GlobalChainProtection_MPS:
//硬线输入定义
Global_ChainProtection_MPS_In:=Global_ChainProtection_MPS_In1 AND Global_ChainProtection_MPS_In2;
//硬线输出定义
Global_ChainProtection_MPS_Out1:=Global_ChainProtection_MPS_Done;
Global_ChainProtection_MPS_Out2:=Global_ChainProtection_MPS_Done;
//总开关
IF NOT Global_ChainProtection_MPS_On THEN
	RETURN;
END_IF
//判断插入件状态，是否就位
//IF NOT IDControlReady THEN
//	Global_ChainProtection_MPS_Done:=FALSE;
//	Error:= TRUE;
//	ErrorID:= 1401;
//	ErrorDescription:='ID NOT READY!';
//	RETURN;
//END_IF
//判断储存环是否给出就位信号，暂时由参数表给出TRUE，最终将由IOC接受PV
IF 	NOT Global_ChainProtection_MPS_StorageRingReady THEN
	Global_ChainProtection_MPS_Done:=FALSE;
	Error:= TRUE;
	ErrorID:= 1403;
	ErrorDescription:='StorageRingChainProtection NOT Ready';
	RETURN;
END_IF
//
//全局连锁保护程序开始
//
//0.检测到下降沿，触发
//1.判断电机是否在开启状态,没有就打开电源
//2.判断是否在Moving状态,若有就Stop
//3.将磁间隙打开到至最大阈值
//4.到位后给出反馈，且安全PLC触发
Global_ChainProtection_MPS_FTRIG(CLK:=Global_ChainProtection_MPS_In);
IF Global_ChainProtection_MPS_FTRIG.Q THEN
	Global_ChainProtection_MPS_Triggered:=TRUE;
END_IF
Global_ChainProtection_MPS_FTRIG_Manul(CLK:=Global_ChainProtection_MPS_ManualOperation);
IF Global_ChainProtection_MPS_FTRIG_Manul.Q THEN
	Global_ChainProtection_MPS_Triggered:=TRUE;
END_IF
IF Global_ChainProtection_MPS_Triggered THEN
	CASE Global_ChainProtection_MPS_State OF
		0://1.判断电机是否在开启状态,没有就打开电源
			IF st_Power=1 THEN
				Global_ChainProtection_MPS_State:=1;
			ELSE
				btn_PowerOn:=TRUE;
				IF btn_PowerOn THEN
					A_PowerOn();
				END_IF
			END_IF
		1://1.判断是否在谱学扫描模式，如果是，则切换回正常运动模式
			IF IsSSMotionMode THEN
				SS_Stop:=TRUE;
				IsSSMotionMode:=FALSE;
			END_IF
			Global_ChainProtection_MPS_State:=2;
		2://判断是否在taper，如果在taper,则判断是否在运动，如果是，则停止运动,0.5sh后，转入下一步
			IF TaperOrNot THEN
				IF moveStatusLeftTop OR moveStatusRightTop OR moveStatusLeftBottom OR moveStatusRightBottom THEN
					btn_UserGapStop:=TRUE;
				ELSE
					Global_ChainProtection_MPS_TON_Stop2Move_InTaperMode(PT:=T#0.5S);
					Global_ChainProtection_MPS_TON_Stop2Move_InTaperMode.IN:=TRUE;
					IF Global_ChainProtection_MPS_TON_Stop2Move_InTaperMode.Q THEN
						TaperOrNot:=FALSE;//关闭taper模式
						Global_ChainProtection_MPS_State:=3;
					END_IF
				END_IF
			ELSE
				Global_ChainProtection_MPS_State:=3;
			END_IF
		3://3.判断是否在Moving状态,若有就Stop.Taper模式已处理完，此处开始走正常GAP开合逻辑
			IF moveStatusLeftTop OR moveStatusRightTop OR moveStatusLeftBottom OR moveStatusRightBottom THEN
				btn_UserGapStop:=TRUE;
			ELSE
				Global_ChainProtection_MPS_TON_Stop2Move(PT:=T#0.5S);
				Global_ChainProtection_MPS_TON_Stop2Move.IN:=TRUE;
				IF Global_ChainProtection_MPS_TON_Stop2Move.Q THEN
					Global_ChainProtection_MPS_State:=4;
				END_IF
			END_IF
		4://当前磁间隙如何和最大磁间隙差别不大，不超过0.1，则直接保护
			IF ABS(UserGapPositionDisplay-Global_ChainProtection_MPS_MaxGapValue)<=0.1 THEN
				Global_ChainProtection_MPS_Done:=TRUE;
				Plc_EmergencyStop:=FALSE;	
				Error:=TRUE;
				ErrorID:=1406;
				ErrorDescription:='MPS Triggered,but ABS(GapPositionDisplay-MPS_MaxGapValue)<=0.1 ';	
			ELSE
				Global_ChainProtection_MPS_State:=5;
			END_IF
		5://5.将磁间隙打开到至最大阈值
			Global_ChainProtection_MPS_TON(PT:=INT_TO_TIME(LREAL_TO_INT(Global_ChainProtection_MPS_MaxGapValue/Global_ChainProtection_MPS_MoveVelocity+30))*1000);
			Global_ChainProtection_MPS_TON.IN:=TRUE;
			Global_ChainProtection_MPS_TON_Power2Move(PT:=T#0.1S);
			Global_ChainProtection_MPS_TON_Power2Move.IN:=TRUE;
			UserGapPositionNew:=Global_ChainProtection_MPS_MaxGapValue;
			UserGapVelocityNew:=Global_ChainProtection_MPS_MoveVelocity;
			btn_UserGapMove:=TRUE;
			IF Global_ChainProtection_MPS_TON_Power2Move.Q THEN
				IF FB_MOVE.BCGapDone THEN
					Global_ChainProtection_MPS_State:=88;
				END_IF
			END_IF
			IF Global_ChainProtection_MPS_TON.Q THEN//如果150s后，还没有运动到指定gap，则报错
				Global_ChainProtection_MPS_State:=-100;
			END_IF
		88://6.到位后给出反馈，且安全PLC触发
			Global_ChainProtection_MPS_Done:=TRUE;
			Plc_EmergencyStop:=FALSE;	
			Error:=TRUE;
			ErrorID:=1404;
			ErrorDescription:='Global_ChainProtection_MPS Triggered ';	
		-100:
			Global_ChainProtection_MPS_Done:=FALSE;
			Error:=TRUE;
			ErrorID:=1405;
			ErrorDescription:='NOT MOVING TO MAXGAP';
	END_CASE
END_IF
END_ACTION

ACTION A_InitCompensationData:
(*补偿开始*)
IF USE_SingleAxis_Compensation THEN
(*正常gap模式以及插入件taper模式下，只运动出口电机，因此只解算出口位置*)
	IF NormalGapMode OR IDTaperMode THEN
		//
		//1.目标位置解算
		//
		(*通过补偿表解算四轴目标位置*)
		//左轴位置由Gap定，右轴位置由右gap定。右gap值=左gap+taper。taper模式和非taper模式一样，非taper模式只是一种特例存在
		//左轴目标位置解算
		IF NOT TaperOrNot THEN
			UserTaperPositionNew:=0;
			//UserTaperPositionDisplay:=0;
		END_IF
		UserRightGapPositionNew:=UserGapPositionNew+UserTaperPositionNew;
		//左轴目标位置解算
		FOR	i:= 1 TO 17 DO
				IF UserGapPositionNew/2<M_Compensation[i+1].Encoder AND UserGapPositionNew/2>=M_Compensation[i].Encoder THEN
					IF i<>18 THEN
						LeftTopLinPositionNew:=(((UserGapPositionNew/2-M_Compensation[i].Encoder)*(M_Compensation[i+1].LeftTop-M_Compensation[i].LeftTop))
								/(M_Compensation[i+1].Encoder-M_Compensation[i].Encoder))+M_Compensation[i].LeftTop;
						LeftBottomLinPositionNew:=(((UserGapPositionNew/2-M_Compensation[i].Encoder)*(M_Compensation[i+1].LeftBottom-M_Compensation[i].LeftBottom))
								/(M_Compensation[i+1].Encoder-M_Compensation[i].Encoder))+M_Compensation[i].LeftBottom;
						M_CompensationNumber:=i;
						InitCompensationDatasDone:=TRUE;
					ELSIF i=18 AND UserGapPositionNew/2=M_Compensation[i].Encoder THEN		(*Gap=14µÄÌØÊâÇé¿ö*)
						(**)
						LeftTopLinPositionNew:=M_Compensation[i].LeftTop;
						LeftBottomLinPositionNew:=M_Compensation[i].LeftBottom;
						M_CompensationNumber:=i;
						InitCompensationDatasDone:=TRUE;
					ELSE
						LeftTopLinPositionNew:=UserGapPositionNew/2;
						LeftBottomLinPositionNew:=UserGapPositionNew/2;
						M_CompensationNumber:=i;
						InitCompensationDatasDone:=TRUE;
					END_IF
				END_IF
		END_FOR
		//右轴目标位置解算
		FOR	j:= 1 TO 17 DO
			IF UserRightGapPositionNew/2<M_Compensation[j+1].Encoder AND UserRightGapPositionNew/2>=M_Compensation[j].Encoder THEN
				IF j<>18 THEN
					RightTopLinPositionNew:=(((UserRightGapPositionNew/2-M_Compensation[j].Encoder)*(M_Compensation[j+1].RightTop-M_Compensation[j].RightTop))
							/(M_Compensation[j+1].Encoder-M_Compensation[j].Encoder))+M_Compensation[j].RightTop;
					RightBottomLinPositionNew:=(((UserRightGapPositionNew/2-M_Compensation[j].Encoder)*(M_Compensation[j+1].RightBottom-M_Compensation[j].RightBottom))
							/(M_Compensation[j+1].Encoder-M_Compensation[j].Encoder))+M_Compensation[j].RightBottom;
					M_CompensationNumber:=j;
					InitCompensationDatasDone:=TRUE;
				ELSIF j=18 AND UserRightGapPositionNew/2=M_Compensation[i].Encoder THEN		(*Gap=14µÄÌØÊâÇé¿ö*)
					(**)
					RightTopLinPositionNew:=M_Compensation[i].RightTop;
					RightBottomLinPositionNew:=M_Compensation[i].RightBottom;
					M_CompensationNumber:=j;
					InitCompensationDatasDone:=TRUE;
				ELSE
					RightTopLinPositionNew:=UserGapPositionNew/2;
					RightBottomLinPositionNew:=UserGapPositionNew/2;
					M_CompensationNumber:=j;
					InitCompensationDatasDone:=TRUE;
				END_IF
			END_IF
		END_FOR
		//
		//2.不论taper还是非taper模式，左轴gap都有左轴发推算，右轴gap由右轴反推算。taper为右gap-左gap
		//
		//左轴显示位置反结算
		FOR k:= 1 TO 17 DO
				IF Pos_LeftTopLin<M_Compensation[k+1].LeftTop AND Pos_LeftTopLin>=M_Compensation[k].LeftTop THEN
					UserGapPositionDisplay_FromLeftTop:=2*(((Pos_LeftTopLin-M_Compensation[k].LeftTop)*(M_Compensation[k+1].Encoder-M_Compensation[k].Encoder))
												/(M_Compensation[k+1].LeftTop-M_Compensation[k].LeftTop)+M_Compensation[k].Encoder);
					UserGapPositionDisplay_FromLeftBottom:=2*(((Pos_LeftBottomLin-M_Compensation[k].LeftBottom)*(M_Compensation[k+1].Encoder-M_Compensation[k].Encoder))
												/(M_Compensation[k+1].LeftBottom-M_Compensation[k].LeftBottom)+M_Compensation[k].Encoder);
					UserGapPositionDisplay:=DINT_TO_LREAL(LREAL_TO_DINT(((UserGapPositionDisplay_FromLeftTop+UserGapPositionDisplay_FromLeftBottom)/2)*100000))/100000;
				END_IF
		END_FOR
		//右轴显示位置反结算
		FOR m:= 1 TO 17 DO
				IF Pos_RightTopLin<M_Compensation[m+1].RightTop AND Pos_RightTopLin>=M_Compensation[m].RightTop THEN
					UserRightGapPositionDisplay_FromRightTop:=2*(((Pos_RightTopLin-M_Compensation[m].RightTop)*(M_Compensation[m+1].Encoder-M_Compensation[m].Encoder))
												/(M_Compensation[m+1].RightTop-M_Compensation[m].RightTop)+M_Compensation[m].Encoder);
					UserRightGapPositionDisplay_FromRightBottom:=2*(((Pos_RightBottomLin-M_Compensation[m].RightBottom)*(M_Compensation[m+1].Encoder-M_Compensation[m].Encoder))
												/(M_Compensation[m+1].RightBottom-M_Compensation[m].RightBottom)+M_Compensation[m].Encoder);
					UserRightGapPositionDisplay:=(UserRightGapPositionDisplay_FromRightTop+UserRightGapPositionDisplay_FromRightBottom)/2;
				END_IF
		END_FOR
		IF TaperOrNot OR (Global_ChainProtection_MPS_Triggered OR Global_ChainProtection_EPS_Triggered)  THEN//安全联锁触发时，需要UserTaperPositionDisplay作为A_MonitoringAllAxis的保护
			UserTaperPositionDisplay:=DINT_TO_LREAL(LREAL_TO_DINT((UserRightGapPositionDisplay-UserGapPositionDisplay)*100000))/100000;
			UserTaperVelocityDisplay:=DINT_TO_LREAL(LREAL_TO_DINT((Velo_RightTopLin+Velo_RightBottomLin)*100000))/100000;
		END_IF
		
		UserTaperPositionDisplayBLSide:=DINT_TO_LREAL(LREAL_TO_DINT((UserTaperPositionDisplay/IDTaperAndBLTaperScale*100000)))/100000;
		
		(*速度可以不用解算，直接用即可*)
		LeftTopLinVelocityDisplay:=Velo_LeftTopLin;
		RightTopLinVelocityDisplay:=Velo_RightTopLin;
		LeftBottomLinVelocityDisplay:=Velo_LeftBottomLin;
		RightBottomLinVelocityDisplay:=Velo_RightBottomLin;
		//Gap velocity
		UserGapVelocityDisplay:=DINT_TO_LREAL(LREAL_TO_DINT(((LeftTopLinVelocityDisplay+RightTopLinVelocityDisplay+
			LeftBottomLinVelocityDisplay+RightBottomLinVelocityDisplay)/2)*100000))/100000;
	
			(*解算单轴位置后，核验并做保护*)
		IF ABS(LeftTopLinPositionNew-UserGapPositionNew/2)>Threshold_motorsTargetPosCalculate THEN
			ErrorID:=1601;
			Error:=TRUE;
			ErrorDescription:='LeftTop Threshold_motorsTargetPosCalculate';
			FB_PlcEmergencyStop();
		END_IF
		//注意右轴解算以UserRightGapPositionNew为基准，考虑到taper
		IF ABS(RightTopLinPositionNew-UserRightGapPositionNew/2)>Threshold_motorsTargetPosCalculate THEN
			ErrorID:=1602;
			Error:=TRUE;
			ErrorDescription:='RightTop Threshold_motorsTargetPosCalculate';
			FB_PlcEmergencyStop();
		END_IF
		IF ABS(LeftBottomLinPositionNew-UserGapPositionNew/2)>Threshold_motorsTargetPosCalculate THEN
			ErrorID:=1603;
			Error:=TRUE;
			ErrorDescription:='LeftBottom Threshold_motorsTargetPosCalculate';
			FB_PlcEmergencyStop();
		END_IF
		//注意右轴解算以UserRightGapPositionNew为基准，考虑到taper
		IF ABS(RightBottomLinPositionNew-UserRightGapPositionNew/2)>Threshold_motorsTargetPosCalculate THEN
			ErrorID:=1604;
			Error:=TRUE;
			ErrorDescription:='RightBottom Threshold_motorsTargetPosCalculate';
			FB_PlcEmergencyStop();
		END_IF
	END_IF
		

(*线站taper模式下，出入口电机位置都解算*)
	IF BLTaperMode THEN
		//
		//1.目标位置解算
		//
		(*通过补偿表解算四轴目标位置*)
		//左轴目标位置解算
		IF NOT BLTaperOrNot THEN
			BLUserTaperPositionNew:=0;
		END_IF
		BLUserLeftGapPositionNew:=UserGapPositionNew-BLUserTaperPositionNew*IDTaperAndBLTaperScale/2;
		BLUserRightGapPositionNew:=UserGapPositionNew+BLUserTaperPositionNew*IDTaperAndBLTaperScale/2;
		//左轴目标位置解算
		FOR	i:= 1 TO 17 DO
				IF BLUserLeftGapPositionNew/2<M_Compensation[i+1].Encoder AND BLUserLeftGapPositionNew/2>=M_Compensation[i].Encoder THEN
					IF i<>18 THEN
						LeftTopLinPositionNew:=(((BLUserLeftGapPositionNew/2-M_Compensation[i].Encoder)*(M_Compensation[i+1].LeftTop-M_Compensation[i].LeftTop))
								/(M_Compensation[i+1].Encoder-M_Compensation[i].Encoder))+M_Compensation[i].LeftTop;
						LeftBottomLinPositionNew:=(((BLUserLeftGapPositionNew/2-M_Compensation[i].Encoder)*(M_Compensation[i+1].LeftBottom-M_Compensation[i].LeftBottom))
								/(M_Compensation[i+1].Encoder-M_Compensation[i].Encoder))+M_Compensation[i].LeftBottom;
						M_CompensationNumber:=i;
						InitCompensationDatasDone:=TRUE;
					ELSIF i=18 AND BLUserLeftGapPositionNew/2=M_Compensation[i].Encoder THEN		(*Gap=14µÄÌØÊâÇé¿ö*)
						(**)
						LeftTopLinPositionNew:=M_Compensation[i].LeftTop;
						LeftBottomLinPositionNew:=M_Compensation[i].LeftBottom;
						M_CompensationNumber:=i;
						InitCompensationDatasDone:=TRUE;
					ELSE
						LeftTopLinPositionNew:=BLUserLeftGapPositionNew/2;
						LeftBottomLinPositionNew:=BLUserLeftGapPositionNew/2;
						M_CompensationNumber:=i;
						InitCompensationDatasDone:=TRUE;
					END_IF
				END_IF
		END_FOR
		//右轴目标位置解算
		FOR	j:= 1 TO 17 DO
			IF BLUserRightGapPositionNew/2<M_Compensation[j+1].Encoder AND BLUserRightGapPositionNew/2>=M_Compensation[j].Encoder THEN
				IF j<>18 THEN
					RightTopLinPositionNew:=(((BLUserRightGapPositionNew/2-M_Compensation[j].Encoder)*(M_Compensation[j+1].RightTop-M_Compensation[j].RightTop))
							/(M_Compensation[j+1].Encoder-M_Compensation[j].Encoder))+M_Compensation[j].RightTop;
					RightBottomLinPositionNew:=(((BLUserRightGapPositionNew/2-M_Compensation[j].Encoder)*(M_Compensation[j+1].RightBottom-M_Compensation[j].RightBottom))
							/(M_Compensation[j+1].Encoder-M_Compensation[j].Encoder))+M_Compensation[j].RightBottom;
					M_CompensationNumber:=j;
					InitCompensationDatasDone:=TRUE;
				ELSIF j=18 AND BLUserRightGapPositionNew/2=M_Compensation[i].Encoder THEN		(*Gap=14µÄÌØÊâÇé¿ö*)
					(**)
					RightTopLinPositionNew:=M_Compensation[i].RightTop;
					RightBottomLinPositionNew:=M_Compensation[i].RightBottom;
					M_CompensationNumber:=j;
					InitCompensationDatasDone:=TRUE;
				ELSE
					RightTopLinPositionNew:=UserGapPositionNew/2;
					RightBottomLinPositionNew:=UserGapPositionNew/2;
					M_CompensationNumber:=j;
					InitCompensationDatasDone:=TRUE;
				END_IF
			END_IF
		END_FOR
		//
		//2.不论taper还是非taper模式，左轴gap都有左轴发推算，右轴gap由右轴反推算。
		//
		//左轴显示位置反结算
		FOR k:= 1 TO 17 DO
				IF Pos_LeftTopLin<M_Compensation[k+1].LeftTop AND Pos_LeftTopLin>=M_Compensation[k].LeftTop THEN
					BLUserGapPositionDisplay_FromLeftTop:=2*(((Pos_LeftTopLin-M_Compensation[k].LeftTop)*(M_Compensation[k+1].Encoder-M_Compensation[k].Encoder))
												/(M_Compensation[k+1].LeftTop-M_Compensation[k].LeftTop)+M_Compensation[k].Encoder);
					BLUserGapPositionDisplay_FromLeftBottom:=2*(((Pos_LeftBottomLin-M_Compensation[k].LeftBottom)*(M_Compensation[k+1].Encoder-M_Compensation[k].Encoder))
												/(M_Compensation[k+1].LeftBottom-M_Compensation[k].LeftBottom)+M_Compensation[k].Encoder);
					BLUserLeftGapPositionDisplay:=DINT_TO_LREAL(LREAL_TO_DINT(((BLUserGapPositionDisplay_FromLeftTop+BLUserGapPositionDisplay_FromLeftBottom)/2)*100000))/100000;
				END_IF
		END_FOR
		//右轴显示位置反结算
		FOR m:= 1 TO 17 DO
				IF Pos_RightTopLin<M_Compensation[m+1].RightTop AND Pos_RightTopLin>=M_Compensation[m].RightTop THEN
					BLUserRightGapPositionDisplay_FromRightTop:=2*(((Pos_RightTopLin-M_Compensation[m].RightTop)*(M_Compensation[m+1].Encoder-M_Compensation[m].Encoder))
												/(M_Compensation[m+1].RightTop-M_Compensation[m].RightTop)+M_Compensation[m].Encoder);
					BLUserRightGapPositionDisplay_FromRightBottom:=2*(((Pos_RightBottomLin-M_Compensation[m].RightBottom)*(M_Compensation[m+1].Encoder-M_Compensation[m].Encoder))
												/(M_Compensation[m+1].RightBottom-M_Compensation[m].RightBottom)+M_Compensation[m].Encoder);
					BLUserRightGapPositionDisplay:=(BLUserRightGapPositionDisplay_FromRightTop+BLUserRightGapPositionDisplay_FromRightBottom)/2;
				END_IF
		END_FOR
		//IF TaperOrNot OR (Global_ChainProtection_MPS_Triggered OR Global_ChainProtection_EPS_Triggered)  THEN//安全联锁触发时，需要UserTaperPositionDisplay作为A_MonitoringAllAxis的保护
		//	UserTaperPositionDisplay:=DINT_TO_LREAL(LREAL_TO_DINT((UserRightGapPositionDisplay-UserGapPositionDisplay)/IDTaperAndBLTaperScale*100000))/100000;
		//	UserTaperVelocityDisplay:=DINT_TO_LREAL(LREAL_TO_DINT((Velo_RightTopLin+Velo_RightBottomLin)/IDTaperAndBLTaperScale/2*100000))/100000;
		//END_IF
		//位置反解算
		UserGapPositionDisplay:=DINT_TO_LREAL(LREAL_TO_DINT(((BLUserLeftGapPositionDisplay+BLUserRightGapPositionDisplay)/2)*100000))/100000;
		BLUserTaperPositionDisplay:=DINT_TO_LREAL(LREAL_TO_DINT(((BLUserRightGapPositionDisplay-BLUserLeftGapPositionDisplay)/IDTaperAndBLTaperScale)*100000))/100000;
		//速度反解算
		LeftTopLinVelocityDisplay:=Velo_LeftTopLin/IDTaperAndBLTaperScale;
		RightTopLinVelocityDisplay:=Velo_RightTopLin/IDTaperAndBLTaperScale;
		LeftBottomLinVelocityDisplay:=Velo_LeftBottomLin/IDTaperAndBLTaperScale;
		RightBottomLinVelocityDisplay:=Velo_RightBottomLin/IDTaperAndBLTaperScale;
		BLUserTaperVelocityDisplay:=DINT_TO_LREAL(LREAL_TO_DINT((RightTopLinVelocityDisplay+RightBottomLinVelocityDisplay-
								(LeftTopLinVelocityDisplay+LeftBottomLinVelocityDisplay))*100000))/100000;
	END_IF

END_IF
END_ACTION

ACTION A_MonitoringAllAxis:
(****************************************************************
NAME:			A_MonitoringAllAxis
DATA:			2018.1.9
VERSION:		1.0.0
DESCRIPTION:	

HISTORY:
				2017.1.9		NEW

***************************************************************)
IF  st_Power<>0 THEN
CASE moni_State OF
0:
		//
		//step1:根据四轴光栅，计算实际位置差和速度差
		//
		(*Top*)
		Diff_UserTopPos_actual:=ABS(Pos_leftTopLin-Pos_RightTopLin);
		(*Bottom*)
		Diff_UserBottomPos_actual:=ABS(Pos_LeftBottomLin-Pos_RightBottomLin);
		(*Left*)
		Diff_UserLeftPos_actual:=ABS(Pos_LeftTopLin-Pos_LeftBottomLin);
		(*Right*)
		Diff_UserRightPos_actual:=ABS(Pos_RightTopLin-Pos_RightBottomLin);
		(*Velocity*)
		(*Top*)
		Diff_UserTopVelo_actual:=ABS(Velo_leftTopLin-Velo_RightTopLin);
		(*Bottom*)
		Diff_UserBottomVelo_actual:=ABS(Velo_LeftBottomLin-Velo_RightBottomLin);
		(*Left*)
		Diff_UserLeftVelo_actual:=ABS(Velo_LeftTopLin-Velo_LeftBottomLin);
		(*Right*)
		Diff_UserRightVelo_actual:=ABS(Velo_RightTopLin-Velo_RightBottomLin);
		//
		//step2:分类计算阈值
		//
		//正常gap模式
		IF NormalGapMode THEN
			Threshold_UserTopPos_PLC:=Threshold_UserTopPos;//位置差=固有阈值，在参数表中调节
			Threshold_UserTopVelo_PLC:=Threshold_UserTopVelo+ABS(UserGapVelocityDisplay);//速度差=固有阈值+当前速度。因为有一轴停止，其它轴还在运动的情况
			Threshold_UserBottomPos_PLC:=Threshold_UserBottomPos;
			Threshold_UserBottomVelo_PLC:=Threshold_UserBottomVelo+ABS(UserGapVelocityDisplay);
			Threshold_UserLeftPos_PLC:=Threshold_UserLeftPos;
			Threshold_UserLeftVelo_PLC:=Threshold_UserLeftVelo+ABS(UserGapVelocityDisplay);
			Threshold_UserRightPos_PLC:=Threshold_UserRightPos;
			Threshold_UserRightVelo_PLC:=Threshold_UserRightVelo+ABS(UserGapVelocityDisplay);
		END_IF		
		//IDTaper模式
		IF IDTaperMode THEN
			Threshold_UserTopPos_PLC:=Threshold_UserTopPos+ABS(UserTaperPositionDisplay*1.1/2);//位置差=固有阈值+当前taper值的一半，1.1为安全系数
			Threshold_UserTopVelo_PLC:=Threshold_UserTopVelo+ABS(UserTaperVelocityDisplay*1.1/2);
			Threshold_UserBottomPos_PLC:=Threshold_UserBottomPos+ABS(UserTaperPositionDisplay*1.1/2);
			Threshold_UserBottomVelo_PLC:=Threshold_UserBottomVelo+ABS(UserTaperVelocityDisplay*1.1/2);
			Threshold_UserLeftPos_PLC:=Threshold_UserLeftPos+ABS(UserTaperPositionDisplay*1.1/2);
			Threshold_UserLeftVelo_PLC:=Threshold_UserLeftVelo+ABS(UserTaperVelocityDisplay*1.1/2);
			Threshold_UserRightPos_PLC:=Threshold_UserRightPos+ABS(UserTaperPositionDisplay*1.1/2);
			Threshold_UserRightVelo_PLC:=Threshold_UserRightVelo+ABS(UserTaperVelocityDisplay*1.1/2);
		END_IF
		//线站taper模式
		IF BLTaperMode THEN
			Threshold_UserTopPos_PLC:=Threshold_UserTopPos+ABS(BLUserTaperPositionDisplay*IDTaperAndBLTaperScale*1.1/2);//Top位置误差=gap运动细微误差+目标taper位置
			Threshold_UserTopVelo_PLC:=Threshold_UserTopVelo+ABS(BLUserTaperVelocityDisplay*IDTaperAndBLTaperScale*1.1/2);//Top速度误差=gap运动细微误差+gap目标速度。因为可能出现一个轴运动完了，另一个轴还在运动的情况
			Threshold_UserBottomPos_PLC:=Threshold_UserBottomPos+ABS(BLUserTaperPositionDisplay*IDTaperAndBLTaperScale*1.1/2);//Bottom同上
			Threshold_UserBottomVelo_PLC:=Threshold_UserBottomVelo+ABS(BLUserTaperVelocityDisplay*IDTaperAndBLTaperScale*1.1/2);
			Threshold_UserLeftPos_PLC:=Threshold_UserLeftPos+ABS(BLUserTaperPositionDisplay*IDTaperAndBLTaperScale*1.1/2);
			Threshold_UserLeftVelo_PLC:=Threshold_UserLeftVelo+ABS(BLUserTaperVelocityDisplay*IDTaperAndBLTaperScale*1.1/2);
			Threshold_UserRightPos_PLC:=Threshold_UserRightPos+ABS(BLUserTaperPositionDisplay*IDTaperAndBLTaperScale*1.1/2);
			Threshold_UserRightVelo_PLC:=Threshold_UserRightVelo+ABS(BLUserTaperVelocityDisplay*IDTaperAndBLTaperScale*1.1/2);
		END_IF
		//
		//step3:保护
		//
		IF Diff_UserTopPos_actual >Threshold_UserTopPos_PLC  THEN
				Error:=TRUE;
				ErrorID:=601;
				ErrorDescription:='Diff_UserTopPos_actual >Threshold_UserTopPos_PLC';
				moni_State:=-100;
		END_IF
		IF Diff_UserTopVelo_actual>Threshold_UserTopVelo_PLC  THEN
				Error:=TRUE;
				ErrorID:=602;
				ErrorDescription:='Diff_UserTopVelo_actual>Threshold_UserTopVelo_PLC';
				moni_State:=-100;
		END_IF
		IF Diff_UserBottomPos_actual>Threshold_UserBottomPos_PLC  THEN
				Error:=TRUE;
				ErrorID:=603;
				ErrorDescription:='Diff_UserBottomPos_actual>Threshold_UserBottomPos_PLC';
				moni_State:=-100;
		END_IF
		IF Diff_UserBottomVelo_actual>Threshold_UserBottomVelo_PLC  THEN
				Error:=TRUE;
				ErrorID:=604;
				ErrorDescription:='Diff_UserBottomVelo_actual>Threshold_UserBottomVelo_PLC';
				moni_State:=-100;
		END_IF
		IF Diff_UserLeftPos_actual>Threshold_UserLeftPos_PLC  THEN
				Error:=TRUE;
				ErrorID:=605;
				ErrorDescription:='Diff_UserLeftPos_actual>Threshold_UserLeftPos_PLC';
				moni_State:=-100;
		END_IF
		IF  Diff_UserLeftVelo_actual>Threshold_UserLeftVelo_PLC THEN
				Error:=TRUE;
				ErrorID:=606;
				ErrorDescription:='Diff_UserLeftVelo_actual>Threshold_UserLeftVelo_PLC';
				moni_State:=-100;	
		END_IF
		IF Diff_UserRightPos_actual>Threshold_UserRightPos_PLC  THEN
				Error:=TRUE;
				ErrorID:=607;
				ErrorDescription:='Diff_UserRightPos_actual>Threshold_UserRightPos_PLC';
				moni_State:=-100;	
		END_IF
		IF  Diff_UserRightVelo_actual>Threshold_UserRightVelo_PLC THEN
				Error:=TRUE;
				ErrorID:=608;
				ErrorDescription:='Diff_UserRightVelo_actual>Threshold_UserRightVelo_PLC';
				moni_State:=-100;
		END_IF
		//单独拿出最大taper来做冗余保护
		IF IDTaperMode THEN
			IF  Diff_UserTopPos_actual > max_UserTaperPositionNew*1.1/2 THEN
					Error:=TRUE;
					ErrorID:=609;
					ErrorDescription:='Diff_UserTopPos_actual > max_UserTaperPositionNew*1.1/2';
					moni_State:=-100;
			END_IF
			IF  Diff_UserBottomPos_actual > max_UserTaperPositionNew*1.1/2 THEN
					Error:=TRUE;
					ErrorID:=610;
					ErrorDescription:='Diff_UserBottomPos_actual > max_UserTaperPositionNew*1.1/2';
					moni_State:=-100;
			END_IF
		END_IF
		IF BLTaperMode THEN
			IF  Diff_UserTopPos_actual > (max_BLUserTaperPositionNew*IDTaperAndBLTaperScale+HysteresisError)*1.1/2 THEN//
					Error:=TRUE;
					ErrorID:=609;
					ErrorDescription:='Diff_UserTopPos_actual > (max_BLUserTaperPositionNew*IDTaperAndBLTaperScale+HysteresisError)*1.1/2';
					moni_State:=-100;
			END_IF
			IF  Diff_UserBottomPos_actual > (max_BLUserTaperPositionNew*IDTaperAndBLTaperScale+HysteresisError)*1.1/2 THEN//
					Error:=TRUE;
					ErrorID:=610;
					ErrorDescription:='Diff_UserBottomPos_actual > (max_BLUserTaperPositionNew*IDTaperAndBLTaperScale+HysteresisError)*1.1/2';
					moni_State:=-100;
			END_IF
		END_IF
-100:
		btn_UserGapStop:=TRUE;
		FB_PlcEmergencyStop();
		Error:=TRUE;
		LED_Error:=TRUE;
END_CASE
END_IF
END_ACTION

ACTION A_OneKeyToMaxGap:
//0.上升沿触发
//1.判断电机是否在开启状态,没有就打开电源
//2.判断是否在Moving状态,若有就Stop
//3.将磁间隙打开到至最大阈值
//4.到位后给出反馈
OneKeyToMaxGap_RTRIG(CLK:=btn_OneKeyToMaxGap);
IF OneKeyToMaxGap_RTRIG.Q THEN
	OneKeyToMaxGap_Triggered:=TRUE;
	OneKeyToMaxGap_Done:=FALSE;
END_IF
IF OneKeyToMaxGap_Triggered THEN
	CASE OneKeyToMaxGap_State OF
		0://1.判断电机是否在开启状态,没有就打开电源
			IF st_Power=1 THEN
				OneKeyToMaxGap_State:=1;
			ELSE
				btn_PowerOn:=TRUE;
				IF btn_PowerOn THEN
					A_PowerOn();
				END_IF
			END_IF
		1://1.判断是否在谱学扫描模式，如果是，则切换回正常运动模式
			IF IsSSMotionMode THEN
				SS_Stop:=TRUE;
				IsSSMotionMode:=FALSE;
			END_IF
			OneKeyToMaxGap_State:=2;
		2://判断是否在taper，如果在taper,则判断是否在运动，如果是，则停止运动,0.5sh后，转入下一步
			IF TaperOrNot THEN
				IF moveStatusLeftTop OR moveStatusRightTop OR moveStatusLeftBottom OR moveStatusRightBottom THEN
					btn_UserGapStop:=TRUE;
				ELSE
					OneKeyToMaxGap_TON_Stop2Move_InTaperMode(PT:=T#0.5S);
					OneKeyToMaxGap_TON_Stop2Move_InTaperMode.IN:=TRUE;
					IF OneKeyToMaxGap_TON_Stop2Move_InTaperMode.Q THEN
						TaperOrNot:=FALSE;//关闭taper模式
						OneKeyToMaxGap_State:=3;
						OneKeyToMaxGap_TON_Stop2Move_InTaperMode.IN:=FALSE;
					END_IF
				END_IF
			ELSE
				OneKeyToMaxGap_State:=3;
			END_IF
		3://3.判断是否在Moving状态,若有就Stop.Taper模式已处理完，此处开始走正常GAP开合逻辑
			IF moveStatusLeftTop OR moveStatusRightTop OR moveStatusLeftBottom OR moveStatusRightBottom THEN
				btn_UserGapStop:=TRUE;
			ELSE
				OneKeyToMaxGap_TON_Stop2Move(PT:=T#0.5S);
				OneKeyToMaxGap_TON_Stop2Move.IN:=TRUE;
				IF OneKeyToMaxGap_TON_Stop2Move.Q THEN
					OneKeyToMaxGap_State:=4;
					OneKeyToMaxGap_TON_Stop2Move.IN:=FALSE;
				END_IF
			END_IF
		4://4.将磁间隙打开到至最大阈值
			OneKeyToMaxGap_TON(PT:=INT_TO_TIME(LREAL_TO_INT(max_UserGapPositionNew+30))*1000);
			OneKeyToMaxGap_TON.IN:=TRUE;
			OneKeyToMaxGap_TON_Power2Move(PT:=T#0.1S);
			OneKeyToMaxGap_TON_Power2Move.IN:=TRUE;
			UserGapPositionNew:=max_UserGapPositionNew;
			UserGapVelocityNew:=1;
			btn_UserGapMove:=TRUE;
			IF OneKeyToMaxGap_TON_Power2Move.Q THEN
				OneKeyToMaxGap_TON_Power2Move.IN:=FALSE;
				IF FB_MOVE.BCGapDone THEN
					OneKeyToMaxGap_State:=88;
				END_IF
			END_IF
			IF OneKeyToMaxGap_TON.Q THEN//如果150s后，还没有运动到指定gap，则报错
				OneKeyToMaxGap_TON.IN:=FALSE;
				OneKeyToMaxGap_State:=-100;
			END_IF
			IF  btn_UserGapStop THEN
				//
				OneKeyToMaxGap_State:=0;
				OneKeyToMaxGap_Triggered:=FALSE;
				btn_OneKeyToMaxGap:=FALSE;
				OneKeyToMaxGap_Triggered:=FALSE;
				OneKeyToMaxGap_State:=0;
			END_IF
		88://6.到位后给出反馈
			OneKeyToMaxGap_Done:=TRUE;	
			Error:=FALSE;
			ErrorID:=0;
			ErrorDescription:='';
			btn_OneKeyToMaxGap:=FALSE;
			OneKeyToMaxGap_Triggered:=FALSE;
			OneKeyToMaxGap_State:=0;
				
		-100:
			OneKeyToMaxGap_Done:=FALSE;
			Error:=TRUE;
			ErrorID:=1705;
			ErrorDescription:='OneKeyToMaxGap Fail';
			btn_OneKeyToMaxGap:=FALSE;
			OneKeyToMaxGap_Triggered:=FALSE;
			OneKeyToMaxGap_State:=0;
	END_CASE
END_IF
END_ACTION

ACTION A_OneKeyToTaperZero:
IF NormalGapMode THEN
	RETURN;
END_IF
//0.上升沿触发
//1.判断当前taper功能是否开启，没有则RETURN
//2.taper=0，目标gap=当前gap,调用btn_GapMove，运动完成
//3.taperOrNot关闭

//0.上升沿触发
OneKeyToTaperZero_RTRIG(CLK:=btn_OneKeyToTaperZero);
IF OneKeyToTaperZero_RTRIG.Q THEN
	OneKeyToTaperZero_Triggered:=TRUE;
	OneKeyToTaperZero_Done:=FALSE;
END_IF
IF IDTaperMode AND UserTaperVelocityNew<>0 THEN
	OneKeyToTaperZero_TON(PT:=INT_TO_TIME(LREAL_TO_INT((CurrentTaperInit+HysteresisError*10)/UserTaperVelocityNew))*1000);
END_IF
IF BLTaperMode AND BLUserTaperVelocityNew<>0 THEN
	OneKeyToTaperZero_TON(PT:=INT_TO_TIME(LREAL_TO_INT((CurrentTaperInit+HysteresisError*20)/BLUserTaperVelocityNew))*1000);
END_IF
OneKeyToTaperZero_Delay(PT:=T#0.5S);
IF OneKeyToTaperZero_Triggered THEN
	CASE OneKeyToTaperZero_State OF
		0://1.判断当前taper功能是否开启，没有则RETURN
			IF IDTaperMode OR BLTaperMode THEN
				OneKeyToTaperZero_State:=1;
			END_IF
		1://2.taper=0，目标gap=当前gap,调用btn_GapMove
			IF IDTaperMode THEN
				UserGapPositionNew:=UserGapPositionDisplay;
				UserTaperPositionNew:=0;
				btn_UserGapMove:=TRUE;
				OneKeyToTaperZero_State:=2;
				IF UserTaperPositionDisplay<=Threshold_TaperChangeFlag THEN//本来当前taper就基本是0,直接关闭taper功能即可
					OneKeyToTaperZero_State:=3;
				END_IF
				CurrentTaperInit:=UserTaperPositionDisplay;
			END_IF
			IF BLTaperMode THEN
				UserGapPositionNew:=UserGapPositionDisplay;
				BLUserTaperPositionNew:=0;
				btn_UserGapMove:=TRUE;
				OneKeyToTaperZero_State:=2;
				IF BLUserTaperPositionDisplay<=Threshold_TaperChangeFlag THEN//本来当前taper就基本是0,直接关闭taper功能即可
					OneKeyToTaperZero_State:=3;
				END_IF
				CurrentTaperInit:=BLUserTaperPositionDisplay;
			END_IF
		2://Move
			OneKeyToTaperZero_TON.IN:=TRUE;
			IF NOT OneKeyToTaperZero_TON.Q THEN
				IF n_state=88 THEN//运动完成
					OneKeyToTaperZero_State:=3;
				END_IF
			ELSE//时间到，还没有运动完，报错
				OneKeyToTaperZero_TON.IN:=FALSE;
				OneKeyToTaperZero_State:=-100;
			END_IF
		3://taper功能关闭
			//延迟0.5s后关闭
			OneKeyToTaperZero_Delay.IN:=TRUE;
			IF OneKeyToTaperZero_Delay.Q THEN
				IF IDTaperMode THEN
					TaperOrNot:=FALSE;
				END_IF
				IF BLTaperMode THEN
					BLTaperOrNot:=FALSE;
				END_IF
				OneKeyToTaperZero_State:=88;				
				OneKeyToTaperZero_Delay.IN:=FALSE;
			END_IF
		88://到位
			OneKeyToTaperZero_Done:=TRUE;	
			Error:=FALSE;
			ErrorID:=0;
			ErrorDescription:='';
			btn_OneKeyToTaperZero:=FALSE;
			OneKeyToTaperZero_Triggered:=FALSE;
			OneKeyToTaperZero_State:=0;
			OneKeyToTaperZero_TON.IN:=FALSE;
			OneKeyToTaperZero_Delay.IN:=FALSE;				
		-100:
			OneKeyToTaperZero_Done:=FALSE;
			Error:=TRUE;
			ErrorID:=1705;
			ErrorDescription:='OneKeyToTaperZero Fail';
			btn_OneKeyToTaperZero:=FALSE;
			OneKeyToTaperZero_Triggered:=FALSE;
			OneKeyToTaperZero_State:=0;
			OneKeyToTaperZero_TON.IN:=FALSE;
	END_CASE
END_IF
END_ACTION

ACTION A_PowerOff:
CASE d_state OF
		0:(*PowerOff*)
			FB_Power(Off:=TRUE);
				d_state:=1;
		1:
			IF NOT FB_power.OffStatus THEN
				d_state:=1;
			ELSE
				d_state:=88;
			END_IF
		88:(*ResetAllState*)
			btn_PowerOn:=FALSE;
			btn_UserGapMove:=FALSE;
			btn_UserGapStop:=FALSE;
			LeftTopLinMoveIndicator:=0;
			RightTopLinMoveIndicator:=0;
			LeftBottomLinMoveIndicator:=0;
			RightBottomLinMoveIndicator:=0;
			fb_ton1.IN:=FALSE;
			fb_ton2.IN:=FALSE;
			fb_ton3.IN:=FALSE;
			State:=0;
			Busy:=FALSE;
			InitPowerDone:=FALSE;
			InitCompensationDatasDone:=FALSE;
			Error:=FALSE;
			ErrorID:=0;
			m_state:=0;
			n_state:=0;
			s_state:=0;
			btn_PowerOff:=FALSE;
			d_state:=0;
			Led_Run:=FALSE;
			Led_Error:=FALSE;
			moni_State:=0;
			i:=0;
END_CASE
END_ACTION

ACTION A_PowerOn:
(****************************************************************
NAME:			A_PowerOn
DATA:			2018.1.9
VERSION:		1.0.0
DESCRIPTION:	

HISTORY:
				2019.1.9		NEW

***************************************************************)
fb_ton3(PT:=t#0.5s);
CASE State OF
	0:	(*FB_Power_On*)
		FB_Power(On:=TRUE);
		fb_ton3.IN:=TRUE;
		State:=1;
	1:	(*wait*)
		FB_power();
		IF NOT FB_power.OnStatus THEN
			IF NOT fb_ton3.Q THEN
				State:=1;
			ELSE
				ErrorID:=1;
				State:=99;
			END_IF
		ELSE
			State:=88;
		END_IF
	88:	(*All Done*)
		btn_PowerOn:=FALSE;
		State:=0;
		Error:=FALSE;
		ErrorID:=0;
		Busy:=FALSE;
		InitPowerDone:=TRUE;
		FB_power.On:=FALSE;
		fb_ton3.IN:=FALSE;
		LED_Error:=FALSE;
	99:
		Error:=TRUE;
		//ErrorID:=701;
		//ErrorDescription:='power on error';		
		btn_PowerOn:=FALSE;
		State:=99;
		Busy:=FALSE;
		InitPowerDone:=FALSE;
		fb_ton3.IN:=FALSE;
		LED_Error:=TRUE;
END_CASE
END_ACTION

ACTION A_RegularMotion:
//Taper运动保护
A_TaperMotionProtection();

(*分别比较四轴目标位置与当前位置的差，如果目标位置比当前位置低，则需要运动到更低-回程差一半；再运动至最终目标位置*)
//只在m=和n=0的时候判断，否则会出现一些BUG，比如往大间隙开时，运动到位后m不能回到0.
IF m_state=0 AND n_state=0 THEN
		TargetPosLessThanCurrentPos:=FALSE;
	IF LeftTopLinPositionNew-Pos_LeftTopLin<-LEDriftErrorThreshold THEN
			TargetPosLessThanCurrentPos:=TRUE;
			TargetLTPosLessThanCurrentLTPos:=TRUE;
	ELSE
				TargetLTPosLessThanCurrentLTPos:=FALSE;
	END_IF
	IF RightTopLinPositionNew-Pos_RightTopLin<-LEDriftErrorThreshold THEN
			TargetPosLessThanCurrentPos:=TRUE;
			TargetRTPosLessThanCurrentRTPos:=TRUE;
	ELSE
			TargetRTPosLessThanCurrentRTPos:=FALSE;
	END_IF
	IF LeftBottomLinPositionNew-Pos_LeftBottomLin<-LEDriftErrorThreshold THEN
			TargetPosLessThanCurrentPos:=TRUE;
			TargetLBPosLessThanCurrentLBPos:=TRUE;
	ELSE
			TargetLBPosLessThanCurrentLBPos:=FALSE;
	END_IF
	IF RightBottomLinPositionNew-Pos_RightBottomLin<-LEDriftErrorThreshold THEN
			TargetPosLessThanCurrentPos:=TRUE;
			TargetRBPosLessThanCurrentRBPos:=TRUE;
	ELSE
			TargetRBPosLessThanCurrentRBPos:=FALSE;
	END_IF
END_IF

(*Move*)
IF InitCompensationDatasDone THEN
		(*四轴目标位置都大于当前位置，直接走到目标位置即可，不需要先走到考虑回城误差的临时位置*)
		IF NOT TargetPosLessThanCurrentPos AND NOT HysteresisMoving THEN
			CASE m_state OF
				0:
					FB_Move.Mode:=5;						//1.gap;2.single;3.taper;4.debug;5.BCGap&UserMode
					FB_Move.CoupleState:=st_Couple;			
					FB_Move.PowerState:=st_Power;						
			
					IF btn_UserGapMove THEN
						IF NOT st_Power THEN
							ErrorID:=1501;
							Error:=TRUE;
							ErrorDescription:='Plz PowerOn Frist';
							LED_Error:=TRUE;
							//btn_UserGapMove:=FALSE;
							RETURN;
						ELSE
							ErrorID:=0;
							Error:=FALSE;
							ErrorDescription:='';
							LED_Error:=FALSE;
							//btn_UserGapMove:=TRUE;
						END_IF
						//目标位置赋值
						FB_Move.BCLeftTopPosition:=LeftTopLinPositionNew;
						FB_Move.BCRightTopPosition:=RightTopLinPositionNew;
						FB_Move.BCLeftBottomPosition:=LeftBottomLinPositionNew;
						FB_Move.BCRightBottomPosition:=RightBottomLinPositionNew;
						//目标速度赋值
						IF NormalGapMode THEN
							FB_Move.BCLeftTopVelocity:=UserGapVelocityNew/2;
							FB_Move.BCRightTopVelocity:=UserGapVelocityNew/2;
							FB_Move.BCLeftBottomVelocity:=UserGapVelocityNew/2;
							FB_Move.BCRightBottomVelocity:=UserGapVelocityNew/2;
						ELSIF IDTaperMode THEN
							FB_Move.BCLeftTopVelocity:=UserTaperVelocityNew/2;
							FB_Move.BCRightTopVelocity:=UserTaperVelocityNew/2;
							FB_Move.BCLeftBottomVelocity:=UserTaperVelocityNew/2;
							FB_Move.BCRightBottomVelocity:=UserTaperVelocityNew/2;
						ELSIF BLTaperMode THEN
							FB_Move.BCLeftTopVelocity:=BLUserTaperVelocityNew*IDTaperAndBLTaperScale/4;
							FB_Move.BCRightTopVelocity:=BLUserTaperVelocityNew*IDTaperAndBLTaperScale/4;
							FB_Move.BCLeftBottomVelocity:=BLUserTaperVelocityNew*IDTaperAndBLTaperScale/4;
							FB_Move.BCRightBottomVelocity:=BLUserTaperVelocityNew*IDTaperAndBLTaperScale/4;
						ELSE
							FB_Move.BCLeftTopVelocity:=0;
							FB_Move.BCRightTopVelocity:=0;
							FB_Move.BCLeftBottomVelocity:=0;
							FB_Move.BCRightBottomVelocity:=0;
						END_IF
						FB_Move.BCGapMove:=TRUE;
						m_state:=1;
						FB_Move();
					END_IF
				1:
					btn_UserGapMove:=FALSE;
					FB_Move();
					IF NOT FB_Move.BCGapDone THEN
						Led_Run:=TRUE;
						m_state:=1;
					ELSE
						m_state:=88;
					END_IF
				88:
					btn_UserGapMove:=FALSE;
					Led_Run:=FALSE;
					m_state:=0;
			END_CASE
		(*四轴有目标位置小于当前位置，先走到临时位置，再走到目标位置*)
		ELSE
			CASE n_state OF
				0:
					FB_Move.Mode:=5;						//1.gap;2.single;3.taper;4.debug;5.BCGap&UserMode;5:userMode_2
					FB_Move.CoupleState:=st_Couple;			
					FB_Move.PowerState:=st_Power;			
					IF btn_UserGapMove THEN	
						IF NOT st_Power THEN
							ErrorID:=1501;
							Error:=TRUE;
							ErrorDescription:='Plz PowerOn Frist';
							LED_Error:=TRUE;
							//btn_UserGapMove:=FALSE;
							RETURN;
						ELSE
							ErrorID:=0;
							Error:=FALSE;
							ErrorDescription:='';
							LED_Error:=FALSE;
							//btn_UserGapMove:=TRUE;
						END_IF						
						//
						IF TargetLTPosLessThanCurrentLTPos THEN			
							FB_Move.BCLeftTopPosition:=LeftTopLinPositionNew-HysteresisError/2;
						ELSE
							FB_Move.BCLeftTopPosition:=LeftTopLinPositionNew;	
						END_IF
						//
						IF TargetRTPosLessThanCurrentRTPos THEN 
							FB_Move.BCRightTopPosition:=RightTopLinPositionNew-HysteresisError/2;
						ELSE					
							FB_Move.BCRightTopPosition:=RightTopLinPositionNew;
						END_IF
						//
						IF TargetLBPosLessThanCurrentLBPos THEN
							FB_Move.BCLeftBottomPosition:=LeftBottomLinPositionNew-HysteresisError/2;
						ELSE
							FB_Move.BCLeftBottomPosition:=LeftBottomLinPositionNew;
						END_IF
						//
						IF TargetRBPosLessThanCurrentRBPos THEN
							FB_Move.BCRightBottomPosition:=RightBottomLinPositionNew-HysteresisError/2;
						ELSE
							FB_Move.BCRightBottomPosition:=RightBottomLinPositionNew;
						END_IF	
						//	close gap情况下，加入了LeftTopLinPositionNewTemp。//
						//如果在往小间隙运行过程中，改变了目标gap，会在第到达第一次目标位置后，继续向第二
						//次输入的目标运动，而不会回到第一次的目标位置。用temp锁定目标位置
						LeftTopLinPositionNewTemp:=LeftTopLinPositionNew;
						RightTopLinPositionNewTemp:=RightTopLinPositionNew;
						LeftBottomLinPositionNewTemp:=LeftBottomLinPositionNew;
						RightBottomLinPositionNewTemp:=RightBottomLinPositionNew;
			
						//
						IF NormalGapMode THEN
							FB_Move.BCLeftTopVelocity:=UserGapVelocityNew/2;
							FB_Move.BCRightTopVelocity:=UserGapVelocityNew/2;
							FB_Move.BCLeftBottomVelocity:=UserGapVelocityNew/2;
							FB_Move.BCRightBottomVelocity:=UserGapVelocityNew/2;
							IF UserGapVelocityNew >1 THEN								  
								ErrorID:=1502;
								Error:=TRUE;
								ErrorDescription:='UserGapVelocityNew must<=1';
								LED_Error:=TRUE;
								btn_UserGapMove:=FALSE;
								RETURN;
							ELSE
								ErrorID:=0;
								Error:=FALSE;
								ErrorDescription:='';
								LED_Error:=FALSE;	
							END_IF									
						ELSIF IDTaperMode THEN
							FB_Move.BCLeftTopVelocity:=UserTaperVelocityNew/2;
							FB_Move.BCRightTopVelocity:=UserTaperVelocityNew/2;
							FB_Move.BCLeftBottomVelocity:=UserTaperVelocityNew/2;
							FB_Move.BCRightBottomVelocity:=UserTaperVelocityNew/2;
						ELSIF BLTaperMode THEN
							FB_Move.BCLeftTopVelocity:=BLUserTaperVelocityNew*IDTaperAndBLTaperScale/4;
							FB_Move.BCRightTopVelocity:=BLUserTaperVelocityNew*IDTaperAndBLTaperScale/4;
							FB_Move.BCLeftBottomVelocity:=BLUserTaperVelocityNew*IDTaperAndBLTaperScale/4;
							FB_Move.BCRightBottomVelocity:=BLUserTaperVelocityNew*IDTaperAndBLTaperScale/4;
						ELSE
							FB_Move.BCLeftTopVelocity:=0;
							FB_Move.BCRightTopVelocity:=0;
							FB_Move.BCLeftBottomVelocity:=0;
							FB_Move.BCRightBottomVelocity:=0;
						END_IF	

